LIN {X 0,Y 573.25,Z 579.072,A -85,B 0,C 180,E1 -2309.824,E2 -2309.824} C_VEL
LIN {X 0,Y 573.282,Z 579.069,A -85,B 0,C 180,E1 -2312.234,E2 -2312.234} C_VEL
LIN {X 0,Y 573.261,Z 579.079,A -85,B 0,C 180,E1 -2315.12,E2 -2315.12} C_VEL
LIN {X 0,Y 573.229,Z 579.076,A -85,B 0,C 180,E1 -2317.662,E2 -2317.662} C_VEL
LIN {X 0,Y 573.247,Z 579.073,A -85,B 0,C 180,E1 -2319.923,E2 -2319.923} C_VEL
LIN {X 0,Y 573.252,Z 579.08,A -85,B 0,C 180,E1 -2322.989,E2 -2322.989} C_VEL
LIN {X 0,Y 573.263,Z 579.072,A -85,B 0,C 180,E1 -2325.806,E2 -2325.806} C_VEL
LIN {X 0,Y 573.273,Z 579.072,A -85,B 0,C 180,E1 -2328.734,E2 -2328.734} C_VEL
LIN {X 0,Y 573.299,Z 579.072,A -85,B 0,C 180,E1 -2331.54,E2 -2331.54} C_VEL
LIN {X 0,Y 573.289,Z 579.067,A -85,B 0,C 180,E1 -2334.371,E2 -2334.371} C_VEL
LIN {X 0,Y 573.299,Z 579.069,A -85,B 0,C 180,E1 -2337.892,E2 -2337.892} C_VEL
LIN {X 0,Y 573.328,Z 579.063,A -85,B 0,C 180,E1 -2340.702,E2 -2340.702} C_VEL
LIN {X 0,Y 573.234,Z 579.085,A -85,B 0,C 180,E1 -2343.514,E2 -2343.514} C_VEL
LIN {X 0,Y 573.283,Z 579.078,A -85,B 0,C 180,E1 -2345.628,E2 -2345.628} C_VEL
LIN {X 0,Y 573.298,Z 579.066,A -85,B 0,C 180,E1 -2348.459,E2 -2348.459} C_VEL
LIN {X 0,Y 573.288,Z 579.072,A -85,B 0,C 180,E1 -2351.311,E2 -2351.311} C_VEL
LIN {X 0,Y 573.269,Z 579.07,A -85,B 0,C 180,E1 -2354.425,E2 -2354.425} C_VEL
LIN {X 0,Y 573.248,Z 579.073,A -85,B 0,C 180,E1 -2357.111,E2 -2357.111} C_VEL
LIN {X 0,Y 573.246,Z 579.079,A -85,B 0,C 180,E1 -2360.076,E2 -2360.076} C_VEL
LIN {X 0,Y 573.227,Z 579.078,A -85,B 0,C 180,E1 -2362.338,E2 -2362.338} C_VEL
LIN {X 0,Y 573.241,Z 579.076,A -85,B 0,C 180,E1 -2364.4,E2 -2364.4} C_VEL
LIN {X 0,Y 572.615,Z 579.154,A -85,B 0,C 180,E1 -2364.986,E2 -2364.986} C_VEL
LIN {X 0,Y 569.777,Z 579.515,A -85,B 0,C 180,E1 -2365.938,E2 -2365.938} C_VEL
LIN {X 0,Y 567.349,Z 579.813,A -85,B 0,C 180,E1 -2366.704,E2 -2366.704} C_VEL
LIN {X 0,Y 566.297,Z 579.94,A -85,B 0,C 180,E1 -2367.295,E2 -2367.295} C_VEL
LIN {X 0,Y 566.207,Z 579.951,A -85,B 0,C 180,E1 -2367.495,E2 -2367.495} C_VEL
LIN {X 0,Y 566.184,Z 579.954,A -85,B 0,C 180,E1 -2370.592,E2 -2370.592} C_VEL
LIN {X 0,Y 566.219,Z 579.948,A -85,B 0,C 180,E1 -2373.102,E2 -2373.102} C_VEL
LIN {X 0,Y 566.202,Z 579.954,A -85,B 0,C 180,E1 -2375.689,E2 -2375.689} C_VEL
LIN {X 0,Y 566.209,Z 579.953,A -85,B 0,C 180,E1 -2378.56,E2 -2378.56} C_VEL
LIN {X 0,Y 566.212,Z 579.949,A -85,B 0,C 180,E1 -2381.136,E2 -2381.136} C_VEL
LIN {X 0,Y 566.192,Z 579.958,A -85,B 0,C 180,E1 -2384.036,E2 -2384.036} C_VEL
LIN {X 0,Y 566.196,Z 579.951,A -85,B 0,C 180,E1 -2387.083,E2 -2387.083} C_VEL
LIN {X 0,Y 566.219,Z 579.95,A -85,B 0,C 180,E1 -2389.803,E2 -2389.803} C_VEL
LIN {X 0,Y 566.192,Z 579.958,A -85,B 0,C 180,E1 -2392.599,E2 -2392.599} C_VEL
LIN {X 0,Y 566.215,Z 579.949,A -85,B 0,C 180,E1 -2395.184,E2 -2395.184} C_VEL
LIN {X 0,Y 566.23,Z 579.947,A -85,B 0,C 180,E1 -2397.744,E2 -2397.744} C_VEL
LIN {X 0,Y 566.199,Z 579.957,A -85,B 0,C 180,E1 -2400.328,E2 -2400.328} C_VEL
LIN {X 0,Y 566.214,Z 579.958,A -85,B 0,C 180,E1 -2402.662,E2 -2402.662} C_VEL
LIN {X 0,Y 566.231,Z 579.95,A -85,B 0,C 180,E1 -2405.039,E2 -2405.039} C_VEL
LIN {X 0,Y 566.191,Z 579.954,A -85,B 0,C 180,E1 -2408.138,E2 -2408.138} C_VEL
LIN {X 0,Y 566.232,Z 579.955,A -85,B 0,C 180,E1 -2410.612,E2 -2410.612} C_VEL
LIN {X 0,Y 566.217,Z 579.95,A -85,B 0,C 180,E1 -2413.413,E2 -2413.413} C_VEL
LIN {X 0,Y 566.198,Z 579.954,A -85,B 0,C 180,E1 -2416.359,E2 -2416.359} C_VEL
LIN {X 0,Y 566.231,Z 579.953,A -85,B 0,C 180,E1 -2418.675,E2 -2418.675} C_VEL
LIN {X 0,Y 566.231,Z 579.949,A -85,B 0,C 180,E1 -2421.435,E2 -2421.435} C_VEL
LIN {X 0,Y 566.261,Z 579.944,A -85,B 0,C 180,E1 -2424.302,E2 -2424.302} C_VEL
LIN {X 0,Y 566.282,Z 579.94,A -85,B 0,C 180,E1 -2427.866,E2 -2427.866} C_VEL
LIN {X 0,Y 566.298,Z 579.942,A -85,B 0,C 180,E1 -2430.711,E2 -2430.711} C_VEL
LIN {X 0,Y 566.27,Z 579.947,A -85,B 0,C 180,E1 -2432.845,E2 -2432.845} C_VEL
LIN {X 0,Y 566.263,Z 579.945,A -85,B 0,C 180,E1 -2435.698,E2 -2435.698} C_VEL
LIN {X 0,Y 566.226,Z 579.948,A -85,B 0,C 180,E1 -2438.566,E2 -2438.566} C_VEL
LIN {X 0,Y 566.239,Z 579.953,A -85,B 0,C 180,E1 -2441.454,E2 -2441.454} C_VEL
LIN {X 0,Y 566.231,Z 579.947,A -85,B 0,C 180,E1 -2444.507,E2 -2444.507} C_VEL
LIN {X 0,Y 566.201,Z 579.96,A -85,B 0,C 180,E1 -2447.331,E2 -2447.331} C_VEL
LIN {X 0,Y 566.21,Z 579.95,A -85,B 0,C 180,E1 -2450.337,E2 -2450.337} C_VEL
LIN {X 0,Y 566.185,Z 579.962,A -85,B 0,C 180,E1 -2453.403,E2 -2453.403} C_VEL
LIN {X 0,Y 566.22,Z 579.958,A -85,B 0,C 180,E1 -2455.748,E2 -2455.748} C_VEL
LIN {X 0,Y 566.26,Z 580.088,A -85,B 0,C 180,E1 -2456.596,E2 -2456.596} C_VEL
LIN {X 0,Y 566.352,Z 587.078,A -85,B 0,C 180,E1 -2457.933,E2 -2457.933} C_VEL
LIN {X 0,Y 566.242,Z 601.154,A -85,B 0,C 180,E1 -2460.588,E2 -2460.588} C_VEL
LIN {X 0,Y 566.228,Z 603.568,A -85,B 0,C 180,E1 -2461.04,E2 -2461.04} C_VEL
LIN {X 0,Y 567.169,Z 609.752,A -85,B 0,C 180,E1 -2461.159,E2 -2461.159} C_VEL
LIN {X 0,Y 566.935,Z 710.865,A -85,B 0,C 180,E1 -2462.465,E2 -2462.465} C_VEL
LIN {X 0,Y 566.836,Z 724.501,A -85,B 0,C 180,E1 -2462.802,E2 -2462.802} C_VEL
LIN {X 0,Y 566.711,Z 737.49,A -85,B 0,C 180,E1 -2463.281,E2 -2463.281} C_VEL
LIN {X 0,Y 566.576,Z 749.083,A -85,B 0,C 180,E1 -2463.862,E2 -2463.862} C_VEL
LIN {X 0,Y 566.403,Z 760.435,A -85,B 0,C 180,E1 -2464.587,E2 -2464.587} C_VEL
LIN {X 0,Y 566.311,Z 770.741,A -85,B 0,C 180,E1 -2465.409,E2 -2465.409} C_VEL
LIN {X 0,Y 566.173,Z 780.385,A -85,B 0,C 180,E1 -2466.364,E2 -2466.364} C_VEL
LIN {X 0,Y 566.044,Z 789.413,A -85,B 0,C 180,E1 -2467.472,E2 -2467.472} C_VEL
LIN {X 0,Y 565.992,Z 796.322,A -85,B 0,C 180,E1 -2468.531,E2 -2468.531} C_VEL
LIN {X 0,Y 565.963,Z 802.163,A -85,B 0,C 180,E1 -2469.656,E2 -2469.656} C_VEL
LIN {X 0,Y 565.922,Z 806.612,A -85,B 0,C 180,E1 -2470.753,E2 -2470.753} C_VEL
LIN {X 0,Y 565.913,Z 810.603,A -85,B 0,C 180,E1 -2472.113,E2 -2472.113} C_VEL
LIN {X 0,Y 565.848,Z 812.476,A -85,B 0,C 180,E1 -2473.086,E2 -2473.086} C_VEL
LIN {X 0,Y 565.843,Z 813.61,A -85,B 0,C 180,E1 -2474.069,E2 -2474.069} C_VEL
LIN {X 0,Y 565.822,Z 813.999,A -85,B 0,C 180,E1 -2475.07,E2 -2475.07} C_VEL
LIN {X 0,Y 565.841,Z 813.567,A -85,B 0,C 180,E1 -2476.085,E2 -2476.085} C_VEL
LIN {X 0,Y 565.858,Z 812.295,A -85,B 0,C 180,E1 -2477.119,E2 -2477.119} C_VEL
LIN {X 0,Y 565.914,Z 810.124,A -85,B 0,C 180,E1 -2478.169,E2 -2478.169} C_VEL
LIN {X 0,Y 565.919,Z 806.927,A -85,B 0,C 180,E1 -2479.246,E2 -2479.246} C_VEL
LIN {X 0,Y 565.962,Z 802.575,A -85,B 0,C 180,E1 -2480.343,E2 -2480.343} C_VEL
LIN {X 0,Y 565.986,Z 796.831,A -85,B 0,C 180,E1 -2481.469,E2 -2481.469} C_VEL
LIN {X 0,Y 566.059,Z 789.431,A -85,B 0,C 180,E1 -2482.616,E2 -2482.616} C_VEL
LIN {X 0,Y 566.161,Z 781.206,A -85,B 0,C 180,E1 -2483.635,E2 -2483.635} C_VEL
LIN {X 0,Y 566.282,Z 772.717,A -85,B 0,C 180,E1 -2484.499,E2 -2484.499} C_VEL
LIN {X 0,Y 566.387,Z 763.144,A -85,B 0,C 180,E1 -2485.303,E2 -2485.303} C_VEL
LIN {X 0,Y 566.546,Z 751.86,A -85,B 0,C 180,E1 -2486.067,E2 -2486.067} C_VEL
LIN {X 0,Y 566.673,Z 739.534,A -85,B 0,C 180,E1 -2486.716,E2 -2486.716} C_VEL
LIN {X 0,Y 566.824,Z 727.276,A -85,B 0,C 180,E1 -2487.2,E2 -2487.2} C_VEL
LIN {X 0,Y 566.908,Z 714.232,A -85,B 0,C 180,E1 -2487.557,E2 -2487.557} C_VEL
LIN {X 0,Y 566.964,Z 698.519,A -85,B 0,C 180,E1 -2487.804,E2 -2487.804} C_VEL
LIN {X 0,Y 567.028,Z 608.635,A -85,B 0,C 180,E1 -2488.948,E2 -2488.948} C_VEL
LIN {X 0,Y 566.211,Z 603.648,A -85,B 0,C 180,E1 -2489.035,E2 -2489.035} C_VEL
LIN {X 0,Y 566.348,Z 589.127,A -85,B 0,C 180,E1 -2491.768,E2 -2491.768} C_VEL
LIN {X 0,Y 566.291,Z 580.244,A -85,B 0,C 180,E1 -2493.463,E2 -2493.463} C_VEL
LIN {X 0,Y 566.235,Z 579.952,A -85,B 0,C 180,E1 -2493.659,E2 -2493.659} C_VEL
LIN {X 0,Y 566.19,Z 579.955,A -85,B 0,C 180,E1 -2495.819,E2 -2495.819} C_VEL
LIN {X 0,Y 566.206,Z 579.956,A -85,B 0,C 180,E1 -2498.903,E2 -2498.903} C_VEL
LIN {X 0,Y 566.204,Z 579.953,A -85,B 0,C 180,E1 -2501.173,E2 -2501.173} C_VEL
LIN {X 0,Y 566.211,Z 579.95,A -85,B 0,C 180,E1 -2503.413,E2 -2503.413} C_VEL
LIN {X 0,Y 566.194,Z 579.957,A -85,B 0,C 180,E1 -2506.359,E2 -2506.359} C_VEL
LIN {X 0,Y 566.264,Z 579.953,A -85,B 0,C 180,E1 -2508.654,E2 -2508.654} C_VEL
LIN {X 0,Y 566.242,Z 579.947,A -85,B 0,C 180,E1 -2511.435,E2 -2511.435} C_VEL
LIN {X 0,Y 566.26,Z 579.946,A -85,B 0,C 180,E1 -2514.302,E2 -2514.302} C_VEL
LIN {X 0,Y 566.271,Z 579.942,A -85,B 0,C 180,E1 -2517.867,E2 -2517.867} C_VEL
LIN {X 0,Y 566.299,Z 579.946,A -85,B 0,C 180,E1 -2520.711,E2 -2520.711} C_VEL
LIN {X 0,Y 566.273,Z 579.951,A -85,B 0,C 180,E1 -2522.846,E2 -2522.846} C_VEL
LIN {X 0,Y 566.261,Z 579.944,A -85,B 0,C 180,E1 -2525.699,E2 -2525.699} C_VEL
LIN {X 0,Y 566.242,Z 579.949,A -85,B 0,C 180,E1 -2528.566,E2 -2528.566} C_VEL
LIN {X 0,Y 566.241,Z 579.949,A -85,B 0,C 180,E1 -2531.455,E2 -2531.455} C_VEL
LIN {X 0,Y 566.224,Z 579.95,A -85,B 0,C 180,E1 -2534.508,E2 -2534.508} C_VEL
LIN {X 0,Y 566.196,Z 579.958,A -85,B 0,C 180,E1 -2537.332,E2 -2537.332} C_VEL
LIN {X 0,Y 566.212,Z 579.949,A -85,B 0,C 180,E1 -2540.338,E2 -2540.338} C_VEL
LIN {X 0,Y 566.182,Z 579.959,A -85,B 0,C 180,E1 -2543.405,E2 -2543.405} C_VEL
LIN {X 0,Y 566.218,Z 579.95,A -85,B 0,C 180,E1 -2545.749,E2 -2545.749} C_VEL
LIN {X 0,Y 566.199,Z 579.95,A -85,B 0,C 180,E1 -2548.204,E2 -2548.204} C_VEL
LIN {X 0,Y 566.188,Z 579.953,A -85,B 0,C 180,E1 -2550.593,E2 -2550.593} C_VEL
LIN {X 0,Y 566.223,Z 579.953,A -85,B 0,C 180,E1 -2553.102,E2 -2553.102} C_VEL
LIN {X 0,Y 566.206,Z 579.954,A -85,B 0,C 180,E1 -2555.689,E2 -2555.689} C_VEL
LIN {X 0,Y 566.213,Z 579.949,A -85,B 0,C 180,E1 -2558.56,E2 -2558.56} C_VEL
LIN {X 0,Y 566.208,Z 579.955,A -85,B 0,C 180,E1 -2561.137,E2 -2561.137} C_VEL
LIN {X 0,Y 566.196,Z 579.953,A -85,B 0,C 180,E1 -2564.036,E2 -2564.036} C_VEL
LIN {X 0,Y 566.198,Z 579.955,A -85,B 0,C 180,E1 -2567.084,E2 -2567.084} C_VEL
LIN {X 0,Y 566.224,Z 579.954,A -85,B 0,C 180,E1 -2569.804,E2 -2569.804} C_VEL
LIN {X 0,Y 566.197,Z 579.951,A -85,B 0,C 180,E1 -2572.6,E2 -2572.6} C_VEL
LIN {X 0,Y 566.219,Z 579.952,A -85,B 0,C 180,E1 -2575.184,E2 -2575.184} C_VEL
LIN {X 0,Y 566.232,Z 579.956,A -85,B 0,C 180,E1 -2577.744,E2 -2577.744} C_VEL
LIN {X 0,Y 566.203,Z 579.953,A -85,B 0,C 180,E1 -2580.329,E2 -2580.329} C_VEL
LIN {X 0,Y 566.212,Z 579.951,A -85,B 0,C 180,E1 -2582.662,E2 -2582.662} C_VEL
LIN {X 0,Y 566.238,Z 579.95,A -85,B 0,C 180,E1 -2585.04,E2 -2585.04} C_VEL
LIN {X 0,Y 566.238,Z 579.992,A -85,B 0,C 180,E1 -2585.848,E2 -2585.848} C_VEL
LIN {X 0,Y 567.17,Z 585.129,A -85,B 0,C 180,E1 -2586.64,E2 -2586.64} C_VEL
LIN {X 0,Y 567.036,Z 601.083,A -85,B 0,C 180,E1 -2588.935,E2 -2588.935} C_VEL
LIN {X 0,Y 566.725,Z 622.357,A -85,B 0,C 180,E1 -2591.94,E2 -2591.94} C_VEL
LIN {X 0,Y 566.453,Z 642.3,A -85,B 0,C 180,E1 -2594.714,E2 -2594.714} C_VEL
LIN {X 0,Y 566.425,Z 651.524,A -85,B 0,C 180,E1 -2595.987,E2 -2595.987} C_VEL
LIN {X 0,Y 567.203,Z 658.268,A -85,B 0,C 180,E1 -2596.096,E2 -2596.096} C_VEL
LIN {X 0,Y 566.978,Z 759.962,A -85,B 0,C 180,E1 -2597.404,E2 -2597.404} C_VEL
LIN {X 0,Y 566.859,Z 772.467,A -85,B 0,C 180,E1 -2597.697,E2 -2597.697} C_VEL
LIN {X 0,Y 566.749,Z 785.381,A -85,B 0,C 180,E1 -2598.149,E2 -2598.149} C_VEL
LIN {X 0,Y 566.627,Z 797.158,A -85,B 0,C 180,E1 -2598.708,E2 -2598.708} C_VEL
LIN {X 0,Y 566.449,Z 809.206,A -85,B 0,C 180,E1 -2599.455,E2 -2599.455} C_VEL
LIN {X 0,Y 566.319,Z 819.603,A -85,B 0,C 180,E1 -2600.266,E2 -2600.266} C_VEL
LIN {X 0,Y 566.207,Z 828.115,A -85,B 0,C 180,E1 -2601.074,E2 -2601.074} C_VEL
LIN {X 0,Y 566.112,Z 835.962,A -85,B 0,C 180,E1 -2601.972,E2 -2601.972} C_VEL
LIN {X 0,Y 566.003,Z 843.622,A -85,B 0,C 180,E1 -2603.047,E2 -2603.047} C_VEL
LIN {X 0,Y 566.004,Z 850.681,A -85,B 0,C 180,E1 -2604.299,E2 -2604.299} C_VEL
LIN {X 0,Y 565.933,Z 855.372,A -85,B 0,C 180,E1 -2605.37,E2 -2605.37} C_VEL
LIN {X 0,Y 565.927,Z 858.957,A -85,B 0,C 180,E1 -2606.44,E2 -2606.44} C_VEL
LIN {X 0,Y 565.878,Z 860.808,A -85,B 0,C 180,E1 -2607.153,E2 -2607.153} C_VEL
LIN {X 0,Y 565.846,Z 863.186,A -85,B 0,C 180,E1 -2608.577,E2 -2608.577} C_VEL
LIN {X 0,Y 565.839,Z 864,A -85,B 0,C 180,E1 -2610,E2 -2610} C_VEL
LIN {X 0,Y 565.846,Z 863.186,A -85,B 0,C 180,E1 -2611.423,E2 -2611.423} C_VEL
LIN {X 0,Y 565.878,Z 860.81,A -85,B 0,C 180,E1 -2612.847,E2 -2612.847} C_VEL
LIN {X 0,Y 565.926,Z 857.896,A -85,B 0,C 180,E1 -2613.916,E2 -2613.916} C_VEL
LIN {X 0,Y 565.878,Z 853.95,A -85,B 0,C 180,E1 -2614.987,E2 -2614.987} C_VEL
LIN {X 0,Y 566.002,Z 848.867,A -85,B 0,C 180,E1 -2616.058,E2 -2616.058} C_VEL
LIN {X 0,Y 566.04,Z 842.47,A -85,B 0,C 180,E1 -2617.132,E2 -2617.132} C_VEL
LIN {X 0,Y 566.134,Z 834.48,A -85,B 0,C 180,E1 -2618.207,E2 -2618.207} C_VEL
LIN {X 0,Y 566.228,Z 826.338,A -85,B 0,C 180,E1 -2619.105,E2 -2619.105} C_VEL
LIN {X 0,Y 566.343,Z 816.404,A -85,B 0,C 180,E1 -2620.005,E2 -2620.005} C_VEL
LIN {X 0,Y 566.524,Z 805.293,A -85,B 0,C 180,E1 -2620.807,E2 -2620.807} C_VEL
LIN {X 0,Y 566.612,Z 794.183,A -85,B 0,C 180,E1 -2621.446,E2 -2621.446} C_VEL
LIN {X 0,Y 566.76,Z 781.992,A -85,B 0,C 180,E1 -2621.987,E2 -2621.987} C_VEL
LIN {X 0,Y 566.875,Z 769.189,A -85,B 0,C 180,E1 -2622.394,E2 -2622.394} C_VEL
LIN {X 0,Y 566.996,Z 755.622,A -85,B 0,C 180,E1 -2622.664,E2 -2622.664} C_VEL
LIN {X 0,Y 567.046,Z 655.806,A -85,B 0,C 180,E1 -2623.939,E2 -2623.939} C_VEL
LIN {X 0,Y 566.424,Z 651.441,A -85,B 0,C 180,E1 -2624.024,E2 -2624.024} C_VEL
LIN {X 0,Y 566.674,Z 627.675,A -85,B 0,C 180,E1 -2627.316,E2 -2627.316} C_VEL
LIN {X 0,Y 566.93,Z 607.733,A -85,B 0,C 180,E1 -2630.12,E2 -2630.12} C_VEL
LIN {X 0,Y 567.238,Z 587.788,A -85,B 0,C 180,E1 -2632.971,E2 -2632.971} C_VEL
LIN {X 0,Y 567.085,Z 584.236,A -85,B 0,C 180,E1 -2633.494,E2 -2633.494} C_VEL
LIN {X 0,Y 566.228,Z 579.955,A -85,B 0,C 180,E1 -2634.179,E2 -2634.179} C_VEL
LIN {X 0,Y 566.209,Z 579.956,A -85,B 0,C 180,E1 -2636.659,E2 -2636.659} C_VEL
LIN {X 0,Y 566.193,Z 579.954,A -85,B 0,C 180,E1 -2638.952,E2 -2638.952} C_VEL
LIN {X 0,Y 566.193,Z 579.952,A -85,B 0,C 180,E1 -2641.421,E2 -2641.421} C_VEL
LIN {X 0,Y 566.212,Z 579.952,A -85,B 0,C 180,E1 -2643.955,E2 -2643.955} C_VEL
LIN {X 0,Y 566.215,Z 579.958,A -85,B 0,C 180,E1 -2646.568,E2 -2646.568} C_VEL
LIN {X 0,Y 566.21,Z 579.949,A -85,B 0,C 180,E1 -2649.685,E2 -2649.685} C_VEL
LIN {X 0,Y 566.207,Z 579.952,A -85,B 0,C 180,E1 -2652.087,E2 -2652.087} C_VEL
LIN {X 0,Y 566.17,Z 579.958,A -85,B 0,C 180,E1 -2655.035,E2 -2655.035} C_VEL
LIN {X 0,Y 566.21,Z 579.949,A -85,B 0,C 180,E1 -2657.912,E2 -2657.912} C_VEL
LIN {X 0,Y 566.218,Z 579.959,A -85,B 0,C 180,E1 -2660.726,E2 -2660.726} C_VEL
LIN {X 0,Y 566.212,Z 579.949,A -85,B 0,C 180,E1 -2663.782,E2 -2663.782} C_VEL
LIN {X 0,Y 566.205,Z 579.951,A -85,B 0,C 180,E1 -2666.265,E2 -2666.265} C_VEL
LIN {X 0,Y 566.197,Z 579.961,A -85,B 0,C 180,E1 -2668.92,E2 -2668.92} C_VEL
LIN {X 0,Y 566.189,Z 579.96,A -85,B 0,C 180,E1 -2671.046,E2 -2671.046} C_VEL
LIN {X 0,Y 566.239,Z 579.948,A -85,B 0,C 180,E1 -2673.46,E2 -2673.46} C_VEL
LIN {X 0,Y 566.191,Z 579.952,A -85,B 0,C 180,E1 -2675.819,E2 -2675.819} C_VEL
LIN {X 0,Y 566.208,Z 579.957,A -85,B 0,C 180,E1 -2678.902,E2 -2678.902} C_VEL
LIN {X 0,Y 566.204,Z 579.96,A -85,B 0,C 180,E1 -2681.172,E2 -2681.172} C_VEL
LIN {X 0,Y 566.211,Z 579.955,A -85,B 0,C 180,E1 -2683.412,E2 -2683.412} C_VEL
LIN {X 0,Y 566.191,Z 579.952,A -85,B 0,C 180,E1 -2686.358,E2 -2686.358} C_VEL
LIN {X 0,Y 566.265,Z 579.944,A -85,B 0,C 180,E1 -2688.653,E2 -2688.653} C_VEL
LIN {X 0,Y 566.24,Z 579.953,A -85,B 0,C 180,E1 -2691.434,E2 -2691.434} C_VEL
LIN {X 0,Y 566.257,Z 579.943,A -85,B 0,C 180,E1 -2694.301,E2 -2694.301} C_VEL
LIN {X 0,Y 566.271,Z 579.945,A -85,B 0,C 180,E1 -2697.866,E2 -2697.866} C_VEL
LIN {X 0,Y 566.298,Z 579.939,A -85,B 0,C 180,E1 -2700.711,E2 -2700.711} C_VEL
LIN {X 0,Y 566.271,Z 579.943,A -85,B 0,C 180,E1 -2702.845,E2 -2702.845} C_VEL
LIN {X 0,Y 566.251,Z 579.952,A -85,B 0,C 180,E1 -2705.698,E2 -2705.698} C_VEL
LIN {X 0,Y 566.239,Z 579.945,A -85,B 0,C 180,E1 -2708.565,E2 -2708.565} C_VEL
LIN {X 0,Y 566.24,Z 579.952,A -85,B 0,C 180,E1 -2711.454,E2 -2711.454} C_VEL
LIN {X 0,Y 566.222,Z 579.948,A -85,B 0,C 180,E1 -2714.507,E2 -2714.507} C_VEL
LIN {X 0,Y 566.193,Z 579.955,A -85,B 0,C 180,E1 -2717.331,E2 -2717.331} C_VEL
LIN {X 0,Y 566.209,Z 579.952,A -85,B 0,C 180,E1 -2720.337,E2 -2720.337} C_VEL
LIN {X 0,Y 566.179,Z 579.956,A -85,B 0,C 180,E1 -2723.404,E2 -2723.404} C_VEL
LIN {X 0,Y 566.215,Z 579.956,A -85,B 0,C 180,E1 -2725.748,E2 -2725.748} C_VEL
LIN {X 0,Y 566.207,Z 579.951,A -85,B 0,C 180,E1 -2727.495,E2 -2727.495} C_VEL
LIN {X 0,Y 565.529,Z 580.042,A -85,B 0,C 180,E1 -2728.089,E2 -2728.089} C_VEL
LIN {X 0,Y 562.663,Z 580.397,A -85,B 0,C 180,E1 -2729.053,E2 -2729.053} C_VEL
LIN {X 0,Y 560.252,Z 580.699,A -85,B 0,C 180,E1 -2729.828,E2 -2729.828} C_VEL
LIN {X 0,Y 559.223,Z 580.823,A -85,B 0,C 180,E1 -2730.427,E2 -2730.427} C_VEL
LIN {X 0,Y 559.143,Z 580.831,A -85,B 0,C 180,E1 -2730.63,E2 -2730.63} C_VEL
LIN {X 0,Y 559.155,Z 580.831,A -85,B 0,C 180,E1 -2733.575,E2 -2733.575} C_VEL
LIN {X 0,Y 559.181,Z 580.829,A -85,B 0,C 180,E1 -2736.452,E2 -2736.452} C_VEL
LIN {X 0,Y 559.17,Z 580.826,A -85,B 0,C 180,E1 -2738.934,E2 -2738.934} C_VEL
LIN {X 0,Y 559.193,Z 580.826,A -85,B 0,C 180,E1 -2741.767,E2 -2741.767} C_VEL
LIN {X 0,Y 559.132,Z 580.834,A -85,B 0,C 180,E1 -2744.739,E2 -2744.739} C_VEL
LIN {X 0,Y 559.155,Z 580.828,A -85,B 0,C 180,E1 -2747.257,E2 -2747.257} C_VEL
LIN {X 0,Y 559.178,Z 580.832,A -85,B 0,C 180,E1 -2750.135,E2 -2750.135} C_VEL
LIN {X 0,Y 559.14,Z 580.833,A -85,B 0,C 180,E1 -2752.893,E2 -2752.893} C_VEL
LIN {X 0,Y 559.155,Z 580.828,A -85,B 0,C 180,E1 -2755.557,E2 -2755.557} C_VEL
LIN {X 0,Y 559.166,Z 580.831,A -85,B 0,C 180,E1 -2758.138,E2 -2758.138} C_VEL
LIN {X 0,Y 559.139,Z 580.839,A -85,B 0,C 180,E1 -2760.647,E2 -2760.647} C_VEL
LIN {X 0,Y 559.166,Z 580.828,A -85,B 0,C 180,E1 -2763.173,E2 -2763.173} C_VEL
LIN {X 0,Y 559.152,Z 580.828,A -85,B 0,C 180,E1 -2765.495,E2 -2765.495} C_VEL
LIN {X 0,Y 559.168,Z 580.836,A -85,B 0,C 180,E1 -2768.624,E2 -2768.624} C_VEL
LIN {X 0,Y 559.167,Z 580.834,A -85,B 0,C 180,E1 -2770.927,E2 -2770.927} C_VEL
LIN {X 0,Y 559.167,Z 580.827,A -85,B 0,C 180,E1 -2773.948,E2 -2773.948} C_VEL
LIN {X 0,Y 559.171,Z 580.827,A -85,B 0,C 180,E1 -2776.184,E2 -2776.184} C_VEL
LIN {X 0,Y 559.191,Z 580.83,A -85,B 0,C 180,E1 -2779.134,E2 -2779.134} C_VEL
LIN {X 0,Y 559.203,Z 580.822,A -85,B 0,C 180,E1 -2782.054,E2 -2782.054} C_VEL
LIN {X 0,Y 559.252,Z 580.826,A -85,B 0,C 180,E1 -2784.953,E2 -2784.953} C_VEL
LIN {X 0,Y 559.253,Z 580.816,A -85,B 0,C 180,E1 -2787.839,E2 -2787.839} C_VEL
LIN {X 0,Y 559.268,Z 580.818,A -85,B 0,C 180,E1 -2790.72,E2 -2790.72} C_VEL
LIN {X 0,Y 559.237,Z 580.824,A -85,B 0,C 180,E1 -2792.881,E2 -2792.881} C_VEL
LIN {X 0,Y 559.231,Z 580.82,A -85,B 0,C 180,E1 -2795.77,E2 -2795.77} C_VEL
LIN {X 0,Y 559.185,Z 580.826,A -85,B 0,C 180,E1 -2798.674,E2 -2798.674} C_VEL
LIN {X 0,Y 559.203,Z 580.827,A -85,B 0,C 180,E1 -2801.6,E2 -2801.6} C_VEL
LIN {X 0,Y 559.196,Z 580.823,A -85,B 0,C 180,E1 -2804.595,E2 -2804.595} C_VEL
LIN {X 0,Y 559.16,Z 580.835,A -85,B 0,C 180,E1 -2807.556,E2 -2807.556} C_VEL
LIN {X 0,Y 559.169,Z 580.831,A -85,B 0,C 180,E1 -2809.837,E2 -2809.837} C_VEL
LIN {X 0,Y 559.138,Z 580.832,A -85,B 0,C 180,E1 -2812.152,E2 -2812.152} C_VEL
LIN {X 0,Y 559.166,Z 580.833,A -85,B 0,C 180,E1 -2815.185,E2 -2815.185} C_VEL
LIN {X 0,Y 559.242,Z 580.929,A -85,B 0,C 180,E1 -2816.519,E2 -2816.519} C_VEL
LIN {X 0,Y 559.333,Z 588.875,A -85,B 0,C 180,E1 -2818.057,E2 -2818.057} C_VEL
LIN {X 0,Y 559.179,Z 603.564,A -85,B 0,C 180,E1 -2820.86,E2 -2820.86} C_VEL
LIN {X 0,Y 560.298,Z 611.174,A -85,B 0,C 180,E1 -2821.004,E2 -2821.004} C_VEL
LIN {X 0,Y 560.023,Z 710.413,A -85,B 0,C 180,E1 -2822.298,E2 -2822.298} C_VEL
LIN {X 0,Y 559.932,Z 723.682,A -85,B 0,C 180,E1 -2822.623,E2 -2822.623} C_VEL
LIN {X 0,Y 559.794,Z 736.752,A -85,B 0,C 180,E1 -2823.102,E2 -2823.102} C_VEL
LIN {X 0,Y 559.634,Z 747.407,A -85,B 0,C 180,E1 -2823.624,E2 -2823.624} C_VEL
LIN {X 0,Y 559.464,Z 758.28,A -85,B 0,C 180,E1 -2824.301,E2 -2824.301} C_VEL
LIN {X 0,Y 559.302,Z 769.442,A -85,B 0,C 180,E1 -2825.174,E2 -2825.174} C_VEL
LIN {X 0,Y 559.151,Z 778.983,A -85,B 0,C 180,E1 -2826.097,E2 -2826.097} C_VEL
LIN {X 0,Y 559.057,Z 787.471,A -85,B 0,C 180,E1 -2827.114,E2 -2827.114} C_VEL
LIN {X 0,Y 558.946,Z 794.928,A -85,B 0,C 180,E1 -2828.215,E2 -2828.215} C_VEL
LIN {X 0,Y 558.886,Z 801.419,A -85,B 0,C 180,E1 -2829.422,E2 -2829.422} C_VEL
LIN {X 0,Y 558.823,Z 805.408,A -85,B 0,C 180,E1 -2830.366,E2 -2830.366} C_VEL
LIN {X 0,Y 558.83,Z 808.779,A -85,B 0,C 180,E1 -2831.379,E2 -2831.379} C_VEL
LIN {X 0,Y 558.815,Z 810.654,A -85,B 0,C 180,E1 -2832.097,E2 -2832.097} C_VEL
LIN {X 0,Y 558.76,Z 812.619,A -85,B 0,C 180,E1 -2833.155,E2 -2833.155} C_VEL
LIN {X 0,Y 558.756,Z 813.703,A -85,B 0,C 180,E1 -2834.198,E2 -2834.198} C_VEL
LIN {X 0,Y 558.741,Z 813.968,A -85,B 0,C 180,E1 -2835.221,E2 -2835.221} C_VEL
LIN {X 0,Y 558.751,Z 813.464,A -85,B 0,C 180,E1 -2836.228,E2 -2836.228} C_VEL
LIN {X 0,Y 558.76,Z 812.18,A -85,B 0,C 180,E1 -2837.219,E2 -2837.219} C_VEL
LIN {X 0,Y 558.814,Z 810.148,A -85,B 0,C 180,E1 -2838.198,E2 -2838.198} C_VEL
LIN {X 0,Y 558.823,Z 807.407,A -85,B 0,C 180,E1 -2839.159,E2 -2839.159} C_VEL
LIN {X 0,Y 558.876,Z 802.873,A -85,B 0,C 180,E1 -2840.343,E2 -2840.343} C_VEL
LIN {X 0,Y 558.921,Z 796.567,A -85,B 0,C 180,E1 -2841.598,E2 -2841.598} C_VEL
LIN {X 0,Y 558.985,Z 789.999,A -85,B 0,C 180,E1 -2842.632,E2 -2842.632} C_VEL
LIN {X 0,Y 559.098,Z 781.814,A -85,B 0,C 180,E1 -2843.675,E2 -2843.675} C_VEL
LIN {X 0,Y 559.254,Z 772.012,A -85,B 0,C 180,E1 -2844.686,E2 -2844.686} C_VEL
LIN {X 0,Y 559.434,Z 761.253,A -85,B 0,C 180,E1 -2845.576,E2 -2845.576} C_VEL
LIN {X 0,Y 559.582,Z 750.402,A -85,B 0,C 180,E1 -2846.292,E2 -2846.292} C_VEL
LIN {X 0,Y 559.716,Z 737.959,A -85,B 0,C 180,E1 -2846.937,E2 -2846.937} C_VEL
LIN {X 0,Y 559.893,Z 724.987,A -85,B 0,C 180,E1 -2847.427,E2 -2847.427} C_VEL
LIN {X 0,Y 559.991,Z 711.747,A -85,B 0,C 180,E1 -2847.766,E2 -2847.766} C_VEL
LIN {X 0,Y 560.101,Z 683.414,A -85,B 0,C 180,E1 -2848.158,E2 -2848.158} C_VEL
LIN {X 0,Y 560.247,Z 610.136,A -85,B 0,C 180,E1 -2849.101,E2 -2849.101} C_VEL
LIN {X 0,Y 559.183,Z 603.625,A -85,B 0,C 180,E1 -2849.219,E2 -2849.219} C_VEL
LIN {X 0,Y 559.319,Z 589.349,A -85,B 0,C 180,E1 -2851.942,E2 -2851.942} C_VEL
LIN {X 0,Y 559.261,Z 581.26,A -85,B 0,C 180,E1 -2853.506,E2 -2853.506} C_VEL
LIN {X 0,Y 559.214,Z 580.827,A -85,B 0,C 180,E1 -2853.604,E2 -2853.604} C_VEL
LIN {X 0,Y 559.147,Z 580.84,A -85,B 0,C 180,E1 -2856.567,E2 -2856.567} C_VEL
LIN {X 0,Y 559.176,Z 580.827,A -85,B 0,C 180,E1 -2859.396,E2 -2859.396} C_VEL
LIN {X 0,Y 559.147,Z 580.83,A -85,B 0,C 180,E1 -2861.686,E2 -2861.686} C_VEL
LIN {X 0,Y 559.162,Z 580.829,A -85,B 0,C 180,E1 -2863.948,E2 -2863.948} C_VEL
LIN {X 0,Y 559.166,Z 580.83,A -85,B 0,C 180,E1 -2866.184,E2 -2866.184} C_VEL
LIN {X 0,Y 559.202,Z 580.827,A -85,B 0,C 180,E1 -2869.134,E2 -2869.134} C_VEL
LIN {X 0,Y 559.205,Z 580.824,A -85,B 0,C 180,E1 -2872.054,E2 -2872.054} C_VEL
LIN {X 0,Y 559.255,Z 580.824,A -85,B 0,C 180,E1 -2874.954,E2 -2874.954} C_VEL
LIN {X 0,Y 559.243,Z 580.818,A -85,B 0,C 180,E1 -2877.84,E2 -2877.84} C_VEL
LIN {X 0,Y 559.268,Z 580.822,A -85,B 0,C 180,E1 -2880.72,E2 -2880.72} C_VEL
LIN {X 0,Y 559.238,Z 580.828,A -85,B 0,C 180,E1 -2882.882,E2 -2882.882} C_VEL
LIN {X 0,Y 559.23,Z 580.819,A -85,B 0,C 180,E1 -2885.771,E2 -2885.771} C_VEL
LIN {X 0,Y 559.197,Z 580.828,A -85,B 0,C 180,E1 -2888.675,E2 -2888.675} C_VEL
LIN {X 0,Y 559.2,Z 580.825,A -85,B 0,C 180,E1 -2891.601,E2 -2891.601} C_VEL
LIN {X 0,Y 559.189,Z 580.827,A -85,B 0,C 180,E1 -2894.596,E2 -2894.596} C_VEL
LIN {X 0,Y 559.155,Z 580.832,A -85,B 0,C 180,E1 -2897.557,E2 -2897.557} C_VEL
LIN {X 0,Y 559.166,Z 580.828,A -85,B 0,C 180,E1 -2899.838,E2 -2899.838} C_VEL
LIN {X 0,Y 559.134,Z 580.83,A -85,B 0,C 180,E1 -2902.153,E2 -2902.153} C_VEL
LIN {X 0,Y 559.172,Z 580.835,A -85,B 0,C 180,E1 -2905.188,E2 -2905.188} C_VEL
LIN {X 0,Y 559.188,Z 580.826,A -85,B 0,C 180,E1 -2907.712,E2 -2907.712} C_VEL
LIN {X 0,Y 559.162,Z 580.827,A -85,B 0,C 180,E1 -2910.183,E2 -2910.183} C_VEL
LIN {X 0,Y 559.169,Z 580.827,A -85,B 0,C 180,E1 -2912.715,E2 -2912.715} C_VEL
LIN {X 0,Y 559.152,Z 580.837,A -85,B 0,C 180,E1 -2915.323,E2 -2915.323} C_VEL
LIN {X 0,Y 559.131,Z 580.832,A -85,B 0,C 180,E1 -2918.018,E2 -2918.018} C_VEL
LIN {X 0,Y 559.172,Z 580.828,A -85,B 0,C 180,E1 -2920.811,E2 -2920.811} C_VEL
LIN {X 0,Y 559.159,Z 580.834,A -85,B 0,C 180,E1 -2923.733,E2 -2923.733} C_VEL
LIN {X 0,Y 559.143,Z 580.831,A -85,B 0,C 180,E1 -2926.804,E2 -2926.804} C_VEL
LIN {X 0,Y 559.173,Z 580.831,A -85,B 0,C 180,E1 -2929.19,E2 -2929.19} C_VEL
LIN {X 0,Y 559.133,Z 580.835,A -85,B 0,C 180,E1 -2931.984,E2 -2931.984} C_VEL
LIN {X 0,Y 559.157,Z 580.829,A -85,B 0,C 180,E1 -2934.679,E2 -2934.679} C_VEL
LIN {X 0,Y 559.173,Z 580.833,A -85,B 0,C 180,E1 -2937.362,E2 -2937.362} C_VEL
LIN {X 0,Y 559.148,Z 580.833,A -85,B 0,C 180,E1 -2940.143,E2 -2940.143} C_VEL
LIN {X 0,Y 559.17,Z 580.83,A -85,B 0,C 180,E1 -2943.098,E2 -2943.098} C_VEL
LIN {X 0,Y 559.205,Z 580.989,A -85,B 0,C 180,E1 -2945.695,E2 -2945.695} C_VEL
LIN {X 0,Y 560.344,Z 587.788,A -85,B 0,C 180,E1 -2946.73,E2 -2946.73} C_VEL
LIN {X 0,Y 560.04,Z 606.402,A -85,B 0,C 180,E1 -2949.429,E2 -2949.429} C_VEL
LIN {X 0,Y 559.707,Z 626.345,A -85,B 0,C 180,E1 -2952.273,E2 -2952.273} C_VEL
LIN {X 0,Y 559.459,Z 646.292,A -85,B 0,C 180,E1 -2955.078,E2 -2955.078} C_VEL
LIN {X 0,Y 559.427,Z 651.524,A -85,B 0,C 180,E1 -2955.808,E2 -2955.808} C_VEL
LIN {X 0,Y 560.326,Z 658.268,A -85,B 0,C 180,E1 -2955.922,E2 -2955.922} C_VEL
LIN {X 0,Y 560.061,Z 759.962,A -85,B 0,C 180,E1 -2957.246,E2 -2957.246} C_VEL
LIN {X 0,Y 559.911,Z 772.467,A -85,B 0,C 180,E1 -2957.542,E2 -2957.542} C_VEL
LIN {X 0,Y 559.801,Z 785.383,A -85,B 0,C 180,E1 -2957.999,E2 -2957.999} C_VEL
LIN {X 0,Y 559.668,Z 796.815,A -85,B 0,C 180,E1 -2958.547,E2 -2958.547} C_VEL
LIN {X 0,Y 559.52,Z 807.913,A -85,B 0,C 180,E1 -2959.232,E2 -2959.232} C_VEL
LIN {X 0,Y 559.31,Z 818.543,A -85,B 0,C 180,E1 -2960.051,E2 -2960.051} C_VEL
LIN {X 0,Y 559.161,Z 828.115,A -85,B 0,C 180,E1 -2960.961,E2 -2960.961} C_VEL
LIN {X 0,Y 559.05,Z 835.962,A -85,B 0,C 180,E1 -2961.87,E2 -2961.87} C_VEL
LIN {X 0,Y 558.944,Z 843.623,A -85,B 0,C 180,E1 -2962.959,E2 -2962.959} C_VEL
LIN {X 0,Y 558.935,Z 850.681,A -85,B 0,C 180,E1 -2964.227,E2 -2964.227} C_VEL
LIN {X 0,Y 558.827,Z 855.373,A -85,B 0,C 180,E1 -2965.311,E2 -2965.311} C_VEL
LIN {X 0,Y 558.837,Z 858.958,A -85,B 0,C 180,E1 -2966.395,E2 -2966.395} C_VEL
LIN {X 0,Y 558.799,Z 860.808,A -85,B 0,C 180,E1 -2967.116,E2 -2967.116} C_VEL
LIN {X 0,Y 558.745,Z 863.185,A -85,B 0,C 180,E1 -2968.559,E2 -2968.559} C_VEL
LIN {X 0,Y 558.74,Z 864,A -85,B 0,C 180,E1 -2970,E2 -2970} C_VEL
LIN {X 0,Y 558.745,Z 863.186,A -85,B 0,C 180,E1 -2971.441,E2 -2971.441} C_VEL
LIN {X 0,Y 558.799,Z 860.81,A -85,B 0,C 180,E1 -2972.884,E2 -2972.884} C_VEL
LIN {X 0,Y 558.844,Z 857.896,A -85,B 0,C 180,E1 -2973.966,E2 -2973.966} C_VEL
LIN {X 0,Y 558.798,Z 853.949,A -85,B 0,C 180,E1 -2975.051,E2 -2975.051} C_VEL
LIN {X 0,Y 558.921,Z 848.868,A -85,B 0,C 180,E1 -2976.135,E2 -2976.135} C_VEL
LIN {X 0,Y 558.977,Z 842.469,A -85,B 0,C 180,E1 -2977.223,E2 -2977.223} C_VEL
LIN {X 0,Y 559.099,Z 834.48,A -85,B 0,C 180,E1 -2978.311,E2 -2978.311} C_VEL
LIN {X 0,Y 559.184,Z 826.338,A -85,B 0,C 180,E1 -2979.221,E2 -2979.221} C_VEL
LIN {X 0,Y 559.355,Z 816.404,A -85,B 0,C 180,E1 -2980.131,E2 -2980.131} C_VEL
LIN {X 0,Y 559.529,Z 805.401,A -85,B 0,C 180,E1 -2980.937,E2 -2980.937} C_VEL
LIN {X 0,Y 559.671,Z 793.468,A -85,B 0,C 180,E1 -2981.627,E2 -2981.627} C_VEL
LIN {X 0,Y 559.85,Z 780.776,A -85,B 0,C 180,E1 -2982.184,E2 -2982.184} C_VEL
LIN {X 0,Y 559.946,Z 767.36,A -85,B 0,C 180,E1 -2982.596,E2 -2982.596} C_VEL
LIN {X 0,Y 560.087,Z 754.107,A -85,B 0,C 180,E1 -2982.846,E2 -2982.846} C_VEL
LIN {X 0,Y 560.227,Z 657.211,A -85,B 0,C 180,E1 -2984.094,E2 -2984.094} C_VEL
LIN {X 0,Y 559.428,Z 651.441,A -85,B 0,C 180,E1 -2984.203,E2 -2984.203} C_VEL
LIN {X 0,Y 559.685,Z 628.794,A -85,B 0,C 180,E1 -2987.381,E2 -2987.381} C_VEL
LIN {X 0,Y 559.992,Z 609.061,A -85,B 0,C 180,E1 -2990.189,E2 -2990.189} C_VEL
LIN {X 0,Y 560.34,Z 589.117,A -85,B 0,C 180,E1 -2993.075,E2 -2993.075} C_VEL
LIN {X 0,Y 560.072,Z 585.113,A -85,B 0,C 180,E1 -2993.674,E2 -2993.674} C_VEL
LIN {X 0,Y 559.193,Z 580.832,A -85,B 0,C 180,E1 -2994.354,E2 -2994.354} C_VEL
LIN {X 0,Y 559.17,Z 580.83,A -85,B 0,C 180,E1 -2996.902,E2 -2996.902} C_VEL
LIN {X 0,Y 559.148,Z 580.833,A -85,B 0,C 180,E1 -2999.857,E2 -2999.857} C_VEL
LIN {X 0,Y 559.175,Z 580.831,A -85,B 0,C 180,E1 -3002.713,E2 -3002.713} C_VEL
LIN {X 0,Y 559.157,Z 580.828,A -85,B 0,C 180,E1 -3005.321,E2 -3005.321} C_VEL
LIN {X 0,Y 559.133,Z 580.833,A -85,B 0,C 180,E1 -3008.016,E2 -3008.016} C_VEL
LIN {X 0,Y 559.173,Z 580.832,A -85,B 0,C 180,E1 -3010.81,E2 -3010.81} C_VEL
LIN {X 0,Y 559.137,Z 580.83,A -85,B 0,C 180,E1 -3013.733,E2 -3013.733} C_VEL
LIN {X 0,Y 559.164,Z 580.835,A -85,B 0,C 180,E1 -3016.8,E2 -3016.8} C_VEL
LIN {X 0,Y 559.172,Z 580.829,A -85,B 0,C 180,E1 -3019.189,E2 -3019.189} C_VEL
LIN {X 0,Y 559.131,Z 580.831,A -85,B 0,C 180,E1 -3021.982,E2 -3021.982} C_VEL
LIN {X 0,Y 559.153,Z 580.838,A -85,B 0,C 180,E1 -3024.782,E2 -3024.782} C_VEL
LIN {X 0,Y 559.168,Z 580.829,A -85,B 0,C 180,E1 -3027.36,E2 -3027.36} C_VEL
LIN {X 0,Y 559.182,Z 580.825,A -85,B 0,C 180,E1 -3030.134,E2 -3030.134} C_VEL
LIN {X 0,Y 559.176,Z 580.832,A -85,B 0,C 180,E1 -3033.169,E2 -3033.169} C_VEL
LIN {X 0,Y 559.149,Z 580.832,A -85,B 0,C 180,E1 -3035.494,E2 -3035.494} C_VEL
LIN {X 0,Y 559.168,Z 580.83,A -85,B 0,C 180,E1 -3038.623,E2 -3038.623} C_VEL
LIN {X 0,Y 559.163,Z 580.834,A -85,B 0,C 180,E1 -3040.926,E2 -3040.926} C_VEL
LIN {X 0,Y 559.161,Z 580.828,A -85,B 0,C 180,E1 -3043.947,E2 -3043.947} C_VEL
LIN {X 0,Y 559.164,Z 580.827,A -85,B 0,C 180,E1 -3046.184,E2 -3046.184} C_VEL
LIN {X 0,Y 559.202,Z 580.83,A -85,B 0,C 180,E1 -3049.133,E2 -3049.133} C_VEL
LIN {X 0,Y 559.201,Z 580.823,A -85,B 0,C 180,E1 -3052.053,E2 -3052.053} C_VEL
LIN {X 0,Y 559.253,Z 580.819,A -85,B 0,C 180,E1 -3054.953,E2 -3054.953} C_VEL
LIN {X 0,Y 559.242,Z 580.821,A -85,B 0,C 180,E1 -3057.839,E2 -3057.839} C_VEL
LIN {X 0,Y 559.268,Z 580.815,A -85,B 0,C 180,E1 -3060.72,E2 -3060.72} C_VEL
LIN {X 0,Y 559.237,Z 580.819,A -85,B 0,C 180,E1 -3062.881,E2 -3062.881} C_VEL
LIN {X 0,Y 559.22,Z 580.827,A -85,B 0,C 180,E1 -3065.77,E2 -3065.77} C_VEL
LIN {X 0,Y 559.194,Z 580.823,A -85,B 0,C 180,E1 -3068.674,E2 -3068.674} C_VEL
LIN {X 0,Y 559.198,Z 580.832,A -85,B 0,C 180,E1 -3071.6,E2 -3071.6} C_VEL
LIN {X 0,Y 559.188,Z 580.824,A -85,B 0,C 180,E1 -3074.595,E2 -3074.595} C_VEL
LIN {X 0,Y 559.153,Z 580.835,A -85,B 0,C 180,E1 -3077.557,E2 -3077.557} C_VEL
LIN {X 0,Y 559.164,Z 580.837,A -85,B 0,C 180,E1 -3079.837,E2 -3079.837} C_VEL
LIN {X 0,Y 559.131,Z 580.836,A -85,B 0,C 180,E1 -3082.153,E2 -3082.153} C_VEL
LIN {X 0,Y 559.168,Z 580.827,A -85,B 0,C 180,E1 -3085.187,E2 -3085.187} C_VEL
LIN {X 0,Y 559.185,Z 580.83,A -85,B 0,C 180,E1 -3087.711,E2 -3087.711} C_VEL
LIN {X 0,Y 559.143,Z 580.831,A -85,B 0,C 180,E1 -3090.63,E2 -3090.63} C_VEL
LIN {X 0,Y 558.479,Z 580.913,A -85,B 0,C 180,E1 -3091.231,E2 -3091.231} C_VEL
LIN {X 0,Y 555.614,Z 581.276,A -85,B 0,C 180,E1 -3092.207,E2 -3092.207} C_VEL
LIN {X 0,Y 553.2,Z 581.573,A -85,B 0,C 180,E1 -3092.993,E2 -3092.993} C_VEL
LIN {X 0,Y 552.179,Z 581.7,A -85,B 0,C 180,E1 -3093.6,E2 -3093.6} C_VEL
LIN {X 0,Y 552.105,Z 581.712,A -85,B 0,C 180,E1 -3093.805,E2 -3093.805} C_VEL
LIN {X 0,Y 552.108,Z 581.707,A -85,B 0,C 180,E1 -3096.746,E2 -3096.746} C_VEL
LIN {X 0,Y 552.126,Z 581.705,A -85,B 0,C 180,E1 -3099.527,E2 -3099.527} C_VEL
LIN {X 0,Y 552.163,Z 581.699,A -85,B 0,C 180,E1 -3101.441,E2 -3101.441} C_VEL
LIN {X 0,Y 552.088,Z 581.714,A -85,B 0,C 180,E1 -3104.532,E2 -3104.532} C_VEL
LIN {X 0,Y 552.123,Z 581.705,A -85,B 0,C 180,E1 -3107.585,E2 -3107.585} C_VEL
LIN {X 0,Y 552.127,Z 581.712,A -85,B 0,C 180,E1 -3110.474,E2 -3110.474} C_VEL
LIN {X 0,Y 552.108,Z 581.706,A -85,B 0,C 180,E1 -3113.316,E2 -3113.316} C_VEL
LIN {X 0,Y 552.134,Z 581.705,A -85,B 0,C 180,E1 -3115.941,E2 -3115.941} C_VEL
LIN {X 0,Y 552.113,Z 581.715,A -85,B 0,C 180,E1 -3118.541,E2 -3118.541} C_VEL
LIN {X 0,Y 552.121,Z 581.704,A -85,B 0,C 180,E1 -3121.438,E2 -3121.438} C_VEL
LIN {X 0,Y 552.125,Z 581.709,A -85,B 0,C 180,E1 -3124.356,E2 -3124.356} C_VEL
LIN {X 0,Y 552.106,Z 581.715,A -85,B 0,C 180,E1 -3126.759,E2 -3126.759} C_VEL
LIN {X 0,Y 552.117,Z 581.708,A -85,B 0,C 180,E1 -3129.12,E2 -3129.12} C_VEL
LIN {X 0,Y 552.127,Z 581.704,A -85,B 0,C 180,E1 -3131.445,E2 -3131.445} C_VEL
LIN {X 0,Y 552.117,Z 581.705,A -85,B 0,C 180,E1 -3133.738,E2 -3133.738} C_VEL
LIN {X 0,Y 552.134,Z 581.703,A -85,B 0,C 180,E1 -3136.005,E2 -3136.005} C_VEL
LIN {X 0,Y 552.159,Z 581.708,A -85,B 0,C 180,E1 -3138.994,E2 -3138.994} C_VEL
LIN {X 0,Y 552.157,Z 581.7,A -85,B 0,C 180,E1 -3141.952,E2 -3141.952} C_VEL
LIN {X 0,Y 552.227,Z 581.7,A -85,B 0,C 180,E1 -3144.889,E2 -3144.889} C_VEL
LIN {X 0,Y 552.224,Z 581.692,A -85,B 0,C 180,E1 -3147.812,E2 -3147.812} C_VEL
LIN {X 0,Y 552.239,Z 581.694,A -85,B 0,C 180,E1 -3150.729,E2 -3150.729} C_VEL
LIN {X 0,Y 552.204,Z 581.701,A -85,B 0,C 180,E1 -3152.918,E2 -3152.918} C_VEL
LIN {X 0,Y 552.199,Z 581.696,A -85,B 0,C 180,E1 -3155.844,E2 -3155.844} C_VEL
LIN {X 0,Y 552.156,Z 581.703,A -85,B 0,C 180,E1 -3158.785,E2 -3158.785} C_VEL
LIN {X 0,Y 552.16,Z 581.702,A -85,B 0,C 180,E1 -3161.75,E2 -3161.75} C_VEL
LIN {X 0,Y 552.133,Z 581.704,A -85,B 0,C 180,E1 -3164.748,E2 -3164.748} C_VEL
LIN {X 0,Y 552.111,Z 581.709,A -85,B 0,C 180,E1 -3167.788,E2 -3167.788} C_VEL
LIN {X 0,Y 552.127,Z 581.706,A -85,B 0,C 180,E1 -3170.101,E2 -3170.101} C_VEL
LIN {X 0,Y 552.092,Z 581.709,A -85,B 0,C 180,E1 -3172.45,E2 -3172.45} C_VEL
LIN {X 0,Y 552.127,Z 581.713,A -85,B 0,C 180,E1 -3175.345,E2 -3175.345} C_VEL
LIN {X 0,Y 552.182,Z 581.839,A -85,B 0,C 180,E1 -3176.453,E2 -3176.453} C_VEL
LIN {X 0,Y 552.324,Z 586.993,A -85,B 0,C 180,E1 -3177.468,E2 -3177.468} C_VEL
LIN {X 0,Y 552.205,Z 600.401,A -85,B 0,C 180,E1 -3180.067,E2 -3180.067} C_VEL
LIN {X 0,Y 552.146,Z 603.617,A -85,B 0,C 180,E1 -3180.685,E2 -3180.685} C_VEL
LIN {X 0,Y 553.381,Z 610.877,A -85,B 0,C 180,E1 -3180.821,E2 -3180.821} C_VEL
LIN {X 0,Y 553.101,Z 709.968,A -85,B 0,C 180,E1 -3182.127,E2 -3182.127} C_VEL
LIN {X 0,Y 552.981,Z 723.201,A -85,B 0,C 180,E1 -3182.45,E2 -3182.45} C_VEL
LIN {X 0,Y 552.806,Z 735.388,A -85,B 0,C 180,E1 -3182.891,E2 -3182.891} C_VEL
LIN {X 0,Y 552.659,Z 747.349,A -85,B 0,C 180,E1 -3183.475,E2 -3183.475} C_VEL
LIN {X 0,Y 552.45,Z 759.057,A -85,B 0,C 180,E1 -3184.219,E2 -3184.219} C_VEL
LIN {X 0,Y 552.256,Z 770.32,A -85,B 0,C 180,E1 -3185.124,E2 -3185.124} C_VEL
LIN {X 0,Y 552.107,Z 779.728,A -85,B 0,C 180,E1 -3186.066,E2 -3186.066} C_VEL
LIN {X 0,Y 551.947,Z 788.959,A -85,B 0,C 180,E1 -3187.215,E2 -3187.215} C_VEL
LIN {X 0,Y 551.858,Z 796.565,A -85,B 0,C 180,E1 -3188.407,E2 -3188.407} C_VEL
LIN {X 0,Y 551.785,Z 802.335,A -85,B 0,C 180,E1 -3189.556,E2 -3189.556} C_VEL
LIN {X 0,Y 551.727,Z 807.461,A -85,B 0,C 180,E1 -3190.894,E2 -3190.894} C_VEL
LIN {X 0,Y 551.74,Z 810.316,A -85,B 0,C 180,E1 -3191.919,E2 -3191.919} C_VEL
LIN {X 0,Y 551.688,Z 811.495,A -85,B 0,C 180,E1 -3192.466,E2 -3192.466} C_VEL
LIN {X 0,Y 551.66,Z 813.056,A -85,B 0,C 180,E1 -3193.466,E2 -3193.466} C_VEL
LIN {X 0,Y 551.66,Z 813.883,A -85,B 0,C 180,E1 -3194.486,E2 -3194.486} C_VEL
LIN {X 0,Y 551.66,Z 813.904,A -85,B 0,C 180,E1 -3195.519,E2 -3195.519} C_VEL
LIN {X 0,Y 551.66,Z 813.12,A -85,B 0,C 180,E1 -3196.564,E2 -3196.564} C_VEL
LIN {X 0,Y 551.695,Z 811.476,A -85,B 0,C 180,E1 -3197.633,E2 -3197.633} C_VEL
LIN {X 0,Y 551.728,Z 808.878,A -85,B 0,C 180,E1 -3198.723,E2 -3198.723} C_VEL
LIN {X 0,Y 551.735,Z 805.19,A -85,B 0,C 180,E1 -3199.841,E2 -3199.841} C_VEL
LIN {X 0,Y 551.826,Z 799.244,A -85,B 0,C 180,E1 -3201.185,E2 -3201.185} C_VEL
LIN {X 0,Y 551.881,Z 792.737,A -85,B 0,C 180,E1 -3202.32,E2 -3202.32} C_VEL
LIN {X 0,Y 552.006,Z 785.561,A -85,B 0,C 180,E1 -3203.329,E2 -3203.329} C_VEL
LIN {X 0,Y 552.167,Z 776.373,A -85,B 0,C 180,E1 -3204.381,E2 -3204.381} C_VEL
LIN {X 0,Y 552.325,Z 766.921,A -85,B 0,C 180,E1 -3205.263,E2 -3205.263} C_VEL
LIN {X 0,Y 552.463,Z 756.154,A -85,B 0,C 180,E1 -3206.073,E2 -3206.073} C_VEL
LIN {X 0,Y 552.707,Z 743.874,A -85,B 0,C 180,E1 -3206.8,E2 -3206.8} C_VEL
LIN {X 0,Y 552.895,Z 731.52,A -85,B 0,C 180,E1 -3207.356,E2 -3207.356} C_VEL
LIN {X 0,Y 552.979,Z 718.07,A -85,B 0,C 180,E1 -3207.785,E2 -3207.785} C_VEL
LIN {X 0,Y 553.135,Z 706.033,A -85,B 0,C 180,E1 -3208.027,E2 -3208.027} C_VEL
LIN {X 0,Y 553.3,Z 610.239,A -85,B 0,C 180,E1 -3209.28,E2 -3209.28} C_VEL
LIN {X 0,Y 552.161,Z 603.569,A -85,B 0,C 180,E1 -3209.414,E2 -3209.414} C_VEL
LIN {X 0,Y 552.292,Z 589.578,A -85,B 0,C 180,E1 -3212.119,E2 -3212.119} C_VEL
LIN {X 0,Y 552.25,Z 582.268,A -85,B 0,C 180,E1 -3213.551,E2 -3213.551} C_VEL
LIN {X 0,Y 552.16,Z 581.706,A -85,B 0,C 180,E1 -3213.699,E2 -3213.699} C_VEL
LIN {X 0,Y 552.1,Z 581.716,A -85,B 0,C 180,E1 -3216.758,E2 -3216.758} C_VEL
LIN {X 0,Y 552.116,Z 581.708,A -85,B 0,C 180,E1 -3219.12,E2 -3219.12} C_VEL
LIN {X 0,Y 552.123,Z 581.706,A -85,B 0,C 180,E1 -3221.445,E2 -3221.445} C_VEL
LIN {X 0,Y 552.111,Z 581.706,A -85,B 0,C 180,E1 -3223.738,E2 -3223.738} C_VEL
LIN {X 0,Y 552.128,Z 581.705,A -85,B 0,C 180,E1 -3226.005,E2 -3226.005} C_VEL
LIN {X 0,Y 552.169,Z 581.705,A -85,B 0,C 180,E1 -3228.994,E2 -3228.994} C_VEL
LIN {X 0,Y 552.158,Z 581.701,A -85,B 0,C 180,E1 -3231.952,E2 -3231.952} C_VEL
LIN {X 0,Y 552.229,Z 581.701,A -85,B 0,C 180,E1 -3234.889,E2 -3234.889} C_VEL
LIN {X 0,Y 552.215,Z 581.693,A -85,B 0,C 180,E1 -3237.812,E2 -3237.812} C_VEL
LIN {X 0,Y 552.238,Z 581.698,A -85,B 0,C 180,E1 -3240.73,E2 -3240.73} C_VEL
LIN {X 0,Y 552.204,Z 581.704,A -85,B 0,C 180,E1 -3242.918,E2 -3242.918} C_VEL
LIN {X 0,Y 552.2,Z 581.695,A -85,B 0,C 180,E1 -3245.844,E2 -3245.844} C_VEL
LIN {X 0,Y 552.164,Z 581.706,A -85,B 0,C 180,E1 -3248.786,E2 -3248.786} C_VEL
LIN {X 0,Y 552.155,Z 581.701,A -85,B 0,C 180,E1 -3251.751,E2 -3251.751} C_VEL
LIN {X 0,Y 552.127,Z 581.709,A -85,B 0,C 180,E1 -3254.749,E2 -3254.749} C_VEL
LIN {X 0,Y 552.107,Z 581.708,A -85,B 0,C 180,E1 -3257.789,E2 -3257.789} C_VEL
LIN {X 0,Y 552.126,Z 581.704,A -85,B 0,C 180,E1 -3260.102,E2 -3260.102} C_VEL
LIN {X 0,Y 552.088,Z 581.709,A -85,B 0,C 180,E1 -3262.451,E2 -3262.451} C_VEL
LIN {X 0,Y 552.149,Z 581.708,A -85,B 0,C 180,E1 -3265.352,E2 -3265.352} C_VEL
LIN {X 0,Y 552.119,Z 581.704,A -85,B 0,C 180,E1 -3268.098,E2 -3268.098} C_VEL
LIN {X 0,Y 552.108,Z 581.707,A -85,B 0,C 180,E1 -3270.609,E2 -3270.609} C_VEL
LIN {X 0,Y 552.123,Z 581.711,A -85,B 0,C 180,E1 -3273.186,E2 -3273.186} C_VEL
LIN {X 0,Y 552.108,Z 581.709,A -85,B 0,C 180,E1 -3275.842,E2 -3275.842} C_VEL
LIN {X 0,Y 552.122,Z 581.709,A -85,B 0,C 180,E1 -3279.063,E2 -3279.063} C_VEL
LIN {X 0,Y 552.136,Z 581.712,A -85,B 0,C 180,E1 -3281.445,E2 -3281.445} C_VEL
LIN {X 0,Y 552.093,Z 581.709,A -85,B 0,C 180,E1 -3284.533,E2 -3284.533} C_VEL
LIN {X 0,Y 552.128,Z 581.713,A -85,B 0,C 180,E1 -3287.585,E2 -3287.585} C_VEL
LIN {X 0,Y 552.132,Z 581.704,A -85,B 0,C 180,E1 -3290.474,E2 -3290.474} C_VEL
LIN {X 0,Y 552.121,Z 581.711,A -85,B 0,C 180,E1 -3293.316,E2 -3293.316} C_VEL
LIN {X 0,Y 552.131,Z 581.71,A -85,B 0,C 180,E1 -3295.94,E2 -3295.94} C_VEL
LIN {X 0,Y 552.119,Z 581.705,A -85,B 0,C 180,E1 -3298.541,E2 -3298.541} C_VEL
LIN {X 0,Y 552.125,Z 581.712,A -85,B 0,C 180,E1 -3301.439,E2 -3301.439} C_VEL
LIN {X 0,Y 552.131,Z 581.709,A -85,B 0,C 180,E1 -3304.357,E2 -3304.357} C_VEL
LIN {X 0,Y 552.161,Z 581.862,A -85,B 0,C 180,E1 -3305.54,E2 -3305.54} C_VEL
LIN {X 0,Y 553.418,Z 589.157,A -85,B 0,C 180,E1 -3306.657,E2 -3306.657} C_VEL
LIN {X 0,Y 553.143,Z 606.402,A -85,B 0,C 180,E1 -3309.161,E2 -3309.161} C_VEL
LIN {X 0,Y 552.769,Z 626.345,A -85,B 0,C 180,E1 -3312.043,E2 -3312.043} C_VEL
LIN {X 0,Y 552.425,Z 647.753,A -85,B 0,C 180,E1 -3315.09,E2 -3315.09} C_VEL
LIN {X 0,Y 552.421,Z 651.535,A -85,B 0,C 180,E1 -3315.626,E2 -3315.626} C_VEL
LIN {X 0,Y 553.422,Z 659.753,A -85,B 0,C 180,E1 -3315.762,E2 -3315.762} C_VEL
LIN {X 0,Y 553.147,Z 759.962,A -85,B 0,C 180,E1 -3317.083,E2 -3317.083} C_VEL
LIN {X 0,Y 552.999,Z 772.466,A -85,B 0,C 180,E1 -3317.383,E2 -3317.383} C_VEL
LIN {X 0,Y 552.85,Z 785.376,A -85,B 0,C 180,E1 -3317.846,E2 -3317.846} C_VEL
LIN {X 0,Y 552.69,Z 797.669,A -85,B 0,C 180,E1 -3318.449,E2 -3318.449} C_VEL
LIN {X 0,Y 552.478,Z 809.202,A -85,B 0,C 180,E1 -3319.186,E2 -3319.186} C_VEL
LIN {X 0,Y 552.269,Z 819.605,A -85,B 0,C 180,E1 -3320.015,E2 -3320.015} C_VEL
LIN {X 0,Y 552.125,Z 828.115,A -85,B 0,C 180,E1 -3320.845,E2 -3320.845} C_VEL
LIN {X 0,Y 552.013,Z 835.962,A -85,B 0,C 180,E1 -3321.765,E2 -3321.765} C_VEL
LIN {X 0,Y 551.889,Z 843.622,A -85,B 0,C 180,E1 -3322.868,E2 -3322.868} C_VEL
LIN {X 0,Y 551.867,Z 850.68,A -85,B 0,C 180,E1 -3324.153,E2 -3324.153} C_VEL
LIN {X 0,Y 551.725,Z 855.373,A -85,B 0,C 180,E1 -3325.251,E2 -3325.251} C_VEL
LIN {X 0,Y 551.751,Z 858.958,A -85,B 0,C 180,E1 -3326.349,E2 -3326.349} C_VEL
LIN {X 0,Y 551.724,Z 860.808,A -85,B 0,C 180,E1 -3327.079,E2 -3327.079} C_VEL
LIN {X 0,Y 551.645,Z 863.185,A -85,B 0,C 180,E1 -3328.54,E2 -3328.54} C_VEL
LIN {X 0,Y 551.64,Z 864,A -85,B 0,C 180,E1 -3330,E2 -3330} C_VEL
LIN {X 0,Y 551.645,Z 863.186,A -85,B 0,C 180,E1 -3331.46,E2 -3331.46} C_VEL
LIN {X 0,Y 551.724,Z 860.81,A -85,B 0,C 180,E1 -3332.921,E2 -3332.921} C_VEL
LIN {X 0,Y 551.764,Z 857.896,A -85,B 0,C 180,E1 -3334.017,E2 -3334.017} C_VEL
LIN {X 0,Y 551.724,Z 853.949,A -85,B 0,C 180,E1 -3335.116,E2 -3335.116} C_VEL
LIN {X 0,Y 551.803,Z 848.192,A -85,B 0,C 180,E1 -3336.341,E2 -3336.341} C_VEL
LIN {X 0,Y 551.926,Z 841.238,A -85,B 0,C 180,E1 -3337.499,E2 -3337.499} C_VEL
LIN {X 0,Y 552.082,Z 832.993,A -85,B 0,C 180,E1 -3338.602,E2 -3338.602} C_VEL
LIN {X 0,Y 552.221,Z 824.541,A -85,B 0,C 180,E1 -3339.523,E2 -3339.523} C_VEL
LIN {X 0,Y 552.425,Z 814.099,A -85,B 0,C 180,E1 -3340.445,E2 -3340.445} C_VEL
LIN {X 0,Y 552.599,Z 803.294,A -85,B 0,C 180,E1 -3341.213,E2 -3341.213} C_VEL
LIN {X 0,Y 552.781,Z 792.414,A -85,B 0,C 180,E1 -3341.83,E2 -3341.83} C_VEL
LIN {X 0,Y 552.93,Z 780.772,A -85,B 0,C 180,E1 -3342.339,E2 -3342.339} C_VEL
LIN {X 0,Y 553.038,Z 767.359,A -85,B 0,C 180,E1 -3342.756,E2 -3342.756} C_VEL
LIN {X 0,Y 553.164,Z 754.107,A -85,B 0,C 180,E1 -3343.01,E2 -3343.01} C_VEL
LIN {X 0,Y 553.256,Z 657.182,A -85,B 0,C 180,E1 -3344.276,E2 -3344.276} C_VEL
LIN {X 0,Y 552.399,Z 651.451,A -85,B 0,C 180,E1 -3344.386,E2 -3344.386} C_VEL
LIN {X 0,Y 552.705,Z 629.488,A -85,B 0,C 180,E1 -3347.508,E2 -3347.508} C_VEL
LIN {X 0,Y 553.051,Z 610.391,A -85,B 0,C 180,E1 -3350.26,E2 -3350.26} C_VEL
LIN {X 0,Y 553.436,Z 590.28,A -85,B 0,C 180,E1 -3353.182,E2 -3353.182} C_VEL
LIN {X 0,Y 553.051,Z 586.155,A -85,B 0,C 180,E1 -3353.8,E2 -3353.8} C_VEL
LIN {X 0,Y 552.151,Z 581.71,A -85,B 0,C 180,E1 -3354.51,E2 -3354.51} C_VEL
LIN {X 0,Y 552.14,Z 581.704,A -85,B 0,C 180,E1 -3357.272,E2 -3357.272} C_VEL
LIN {X 0,Y 552.117,Z 581.711,A -85,B 0,C 180,E1 -3360.05,E2 -3360.05} C_VEL
LIN {X 0,Y 552.128,Z 581.707,A -85,B 0,C 180,E1 -3362.848,E2 -3362.848} C_VEL
LIN {X 0,Y 552.106,Z 581.706,A -85,B 0,C 180,E1 -3365.443,E2 -3365.443} C_VEL
LIN {X 0,Y 552.096,Z 581.709,A -85,B 0,C 180,E1 -3367.885,E2 -3367.885} C_VEL
LIN {X 0,Y 552.139,Z 581.711,A -85,B 0,C 180,E1 -3370.477,E2 -3370.477} C_VEL
LIN {X 0,Y 552.115,Z 581.705,A -85,B 0,C 180,E1 -3373.484,E2 -3373.484} C_VEL
LIN {X 0,Y 552.116,Z 581.714,A -85,B 0,C 180,E1 -3376.577,E2 -3376.577} C_VEL
LIN {X 0,Y 552.118,Z 581.705,A -85,B 0,C 180,E1 -3379.519,E2 -3379.519} C_VEL
LIN {X 0,Y 552.089,Z 581.711,A -85,B 0,C 180,E1 -3382.335,E2 -3382.335} C_VEL
LIN {X 0,Y 552.122,Z 581.71,A -85,B 0,C 180,E1 -3385.053,E2 -3385.053} C_VEL
LIN {X 0,Y 552.121,Z 581.704,A -85,B 0,C 180,E1 -3387.681,E2 -3387.681} C_VEL
LIN {X 0,Y 552.138,Z 581.703,A -85,B 0,C 180,E1 -3390.236,E2 -3390.236} C_VEL
LIN {X 0,Y 552.14,Z 581.712,A -85,B 0,C 180,E1 -3392.997,E2 -3392.997} C_VEL
LIN {X 0,Y 552.106,Z 581.714,A -85,B 0,C 180,E1 -3395.161,E2 -3395.161} C_VEL
LIN {X 0,Y 552.088,Z 581.711,A -85,B 0,C 180,E1 -3397.548,E2 -3397.548} C_VEL
LIN {X 0,Y 552.14,Z 581.703,A -85,B 0,C 180,E1 -3400.372,E2 -3400.372} C_VEL
LIN {X 0,Y 552.148,Z 581.708,A -85,B 0,C 180,E1 -3402.977,E2 -3402.977} C_VEL
LIN {X 0,Y 552.127,Z 581.704,A -85,B 0,C 180,E1 -3406.004,E2 -3406.004} C_VEL
LIN {X 0,Y 552.169,Z 581.704,A -85,B 0,C 180,E1 -3408.993,E2 -3408.993} C_VEL
LIN {X 0,Y 552.155,Z 581.701,A -85,B 0,C 180,E1 -3411.951,E2 -3411.951} C_VEL
LIN {X 0,Y 552.227,Z 581.694,A -85,B 0,C 180,E1 -3414.889,E2 -3414.889} C_VEL
LIN {X 0,Y 552.214,Z 581.696,A -85,B 0,C 180,E1 -3417.811,E2 -3417.811} C_VEL
LIN {X 0,Y 552.237,Z 581.69,A -85,B 0,C 180,E1 -3420.729,E2 -3420.729} C_VEL
LIN {X 0,Y 552.203,Z 581.696,A -85,B 0,C 180,E1 -3422.918,E2 -3422.918} C_VEL
LIN {X 0,Y 552.19,Z 581.701,A -85,B 0,C 180,E1 -3425.844,E2 -3425.844} C_VEL
LIN {X 0,Y 552.162,Z 581.699,A -85,B 0,C 180,E1 -3428.785,E2 -3428.785} C_VEL
LIN {X 0,Y 552.154,Z 581.709,A -85,B 0,C 180,E1 -3431.75,E2 -3431.75} C_VEL
LIN {X 0,Y 552.125,Z 581.704,A -85,B 0,C 180,E1 -3434.748,E2 -3434.748} C_VEL
LIN {X 0,Y 552.104,Z 581.717,A -85,B 0,C 180,E1 -3437.788,E2 -3437.788} C_VEL
LIN {X 0,Y 552.123,Z 581.709,A -85,B 0,C 180,E1 -3440.101,E2 -3440.101} C_VEL
LIN {X 0,Y 552.085,Z 581.71,A -85,B 0,C 180,E1 -3442.451,E2 -3442.451} C_VEL
LIN {X 0,Y 552.146,Z 581.703,A -85,B 0,C 180,E1 -3445.351,E2 -3445.351} C_VEL
LIN {X 0,Y 552.117,Z 581.713,A -85,B 0,C 180,E1 -3448.097,E2 -3448.097} C_VEL
LIN {X 0,Y 552.103,Z 581.708,A -85,B 0,C 180,E1 -3450.625,E2 -3450.625} C_VEL
LIN {X 0,Y 552.113,Z 581.705,A -85,B 0,C 180,E1 -3453.186,E2 -3453.186} C_VEL
LIN {X 0,Y 552.105,Z 581.712,A -85,B 0,C 180,E1 -3453.805,E2 -3453.805} C_VEL
LIN {X 0,Y 551.471,Z 581.797,A -85,B 0,C 180,E1 -3454.414,E2 -3454.414} C_VEL
LIN {X 0,Y 548.651,Z 582.147,A -85,B 0,C 180,E1 -3455.402,E2 -3455.402} C_VEL
LIN {X 0,Y 546.231,Z 582.447,A -85,B 0,C 180,E1 -3456.198,E2 -3456.198} C_VEL
LIN {X 0,Y 545.161,Z 582.573,A -85,B 0,C 180,E1 -3456.811,E2 -3456.811} C_VEL
LIN {X 0,Y 545.058,Z 582.584,A -85,B 0,C 180,E1 -3457.019,E2 -3457.019} C_VEL
LIN {X 0,Y 545.085,Z 582.59,A -85,B 0,C 180,E1 -3460.14,E2 -3460.14} C_VEL
LIN {X 0,Y 545.059,Z 582.587,A -85,B 0,C 180,E1 -3462.698,E2 -3462.698} C_VEL
LIN {X 0,Y 545.055,Z 582.585,A -85,B 0,C 180,E1 -3465.167,E2 -3465.167} C_VEL
LIN {X 0,Y 545.075,Z 582.585,A -85,B 0,C 180,E1 -3467.898,E2 -3467.898} C_VEL
LIN {X 0,Y 545.077,Z 582.585,A -85,B 0,C 180,E1 -3470.819,E2 -3470.819} C_VEL
LIN {X 0,Y 545.049,Z 582.586,A -85,B 0,C 180,E1 -3473.621,E2 -3473.621} C_VEL
LIN {X 0,Y 545.072,Z 582.59,A -85,B 0,C 180,E1 -3476.33,E2 -3476.33} C_VEL
LIN {X 0,Y 545.062,Z 582.587,A -85,B 0,C 180,E1 -3478.953,E2 -3478.953} C_VEL
LIN {X 0,Y 545.099,Z 582.579,A -85,B 0,C 180,E1 -3481.508,E2 -3481.508} C_VEL
LIN {X 0,Y 545.09,Z 582.588,A -85,B 0,C 180,E1 -3484.491,E2 -3484.491} C_VEL
LIN {X 0,Y 545.04,Z 582.588,A -85,B 0,C 180,E1 -3487.243,E2 -3487.243} C_VEL
LIN {X 0,Y 545.117,Z 582.582,A -85,B 0,C 180,E1 -3490.415,E2 -3490.415} C_VEL
LIN {X 0,Y 545.073,Z 582.583,A -85,B 0,C 180,E1 -3493.522,E2 -3493.522} C_VEL
LIN {X 0,Y 545.093,Z 582.58,A -85,B 0,C 180,E1 -3495.82,E2 -3495.82} C_VEL
LIN {X 0,Y 545.115,Z 582.587,A -85,B 0,C 180,E1 -3498.85,E2 -3498.85} C_VEL
LIN {X 0,Y 545.128,Z 582.575,A -85,B 0,C 180,E1 -3501.847,E2 -3501.847} C_VEL
LIN {X 0,Y 545.203,Z 582.573,A -85,B 0,C 180,E1 -3504.823,E2 -3504.823} C_VEL
LIN {X 0,Y 545.195,Z 582.568,A -85,B 0,C 180,E1 -3507.784,E2 -3507.784} C_VEL
LIN {X 0,Y 545.209,Z 582.57,A -85,B 0,C 180,E1 -3510.739,E2 -3510.739} C_VEL
LIN {X 0,Y 545.171,Z 582.577,A -85,B 0,C 180,E1 -3512.956,E2 -3512.956} C_VEL
LIN {X 0,Y 545.169,Z 582.571,A -85,B 0,C 180,E1 -3515.919,E2 -3515.919} C_VEL
LIN {X 0,Y 545.115,Z 582.581,A -85,B 0,C 180,E1 -3518.9,E2 -3518.9} C_VEL
LIN {X 0,Y 545.132,Z 582.576,A -85,B 0,C 180,E1 -3521.904,E2 -3521.904} C_VEL
LIN {X 0,Y 545.083,Z 582.585,A -85,B 0,C 180,E1 -3524.943,E2 -3524.943} C_VEL
LIN {X 0,Y 545.079,Z 582.583,A -85,B 0,C 180,E1 -3528.025,E2 -3528.025} C_VEL
LIN {X 0,Y 545.092,Z 582.581,A -85,B 0,C 180,E1 -3530.372,E2 -3530.372} C_VEL
LIN {X 0,Y 545.087,Z 582.591,A -85,B 0,C 180,E1 -3533.558,E2 -3533.558} C_VEL
LIN {X 0,Y 545.147,Z 582.639,A -85,B 0,C 180,E1 -3536.356,E2 -3536.356} C_VEL
LIN {X 0,Y 545.317,Z 587.808,A -85,B 0,C 180,E1 -3537.396,E2 -3537.396} C_VEL
LIN {X 0,Y 545.17,Z 602.002,A -85,B 0,C 180,E1 -3540.182,E2 -3540.182} C_VEL
LIN {X 0,Y 545.114,Z 603.639,A -85,B 0,C 180,E1 -3540.5,E2 -3540.5} C_VEL
LIN {X 0,Y 546.538,Z 613.023,A -85,B 0,C 180,E1 -3540.668,E2 -3540.668} C_VEL
LIN {X 0,Y 546.204,Z 710.282,A -85,B 0,C 180,E1 -3541.967,E2 -3541.967} C_VEL
LIN {X 0,Y 546.038,Z 723.551,A -85,B 0,C 180,E1 -3542.298,E2 -3542.298} C_VEL
LIN {X 0,Y 545.88,Z 735.341,A -85,B 0,C 180,E1 -3542.733,E2 -3542.733} C_VEL
LIN {X 0,Y 545.686,Z 747.561,A -85,B 0,C 180,E1 -3543.337,E2 -3543.337} C_VEL
LIN {X 0,Y 545.457,Z 759.18,A -85,B 0,C 180,E1 -3544.088,E2 -3544.088} C_VEL
LIN {X 0,Y 545.235,Z 770.385,A -85,B 0,C 180,E1 -3545.001,E2 -3545.001} C_VEL
LIN {X 0,Y 545.056,Z 780.192,A -85,B 0,C 180,E1 -3546.003,E2 -3546.003} C_VEL
LIN {X 0,Y 544.905,Z 788.728,A -85,B 0,C 180,E1 -3547.081,E2 -3547.081} C_VEL
LIN {X 0,Y 544.786,Z 796.226,A -85,B 0,C 180,E1 -3548.258,E2 -3548.258} C_VEL
LIN {X 0,Y 544.733,Z 801.427,A -85,B 0,C 180,E1 -3549.277,E2 -3549.277} C_VEL
LIN {X 0,Y 544.629,Z 806.055,A -85,B 0,C 180,E1 -3550.418,E2 -3550.418} C_VEL
LIN {X 0,Y 544.652,Z 809.521,A -85,B 0,C 180,E1 -3551.548,E2 -3551.548} C_VEL
LIN {X 0,Y 544.587,Z 811.903,A -85,B 0,C 180,E1 -3552.643,E2 -3552.643} C_VEL
LIN {X 0,Y 544.551,Z 813.705,A -85,B 0,C 180,E1 -3554.18,E2 -3554.18} C_VEL
LIN {X 0,Y 544.548,Z 813.969,A -85,B 0,C 180,E1 -3555.22,E2 -3555.22} C_VEL
LIN {X 0,Y 544.559,Z 813.444,A -85,B 0,C 180,E1 -3556.279,E2 -3556.279} C_VEL
LIN {X 0,Y 544.586,Z 812.057,A -85,B 0,C 180,E1 -3557.356,E2 -3557.356} C_VEL
LIN {X 0,Y 544.627,Z 808.67,A -85,B 0,C 180,E1 -3558.844,E2 -3558.844} C_VEL
LIN {X 0,Y 544.658,Z 805.501,A -85,B 0,C 180,E1 -3559.822,E2 -3559.822} C_VEL
LIN {X 0,Y 544.706,Z 800.41,A -85,B 0,C 180,E1 -3561.025,E2 -3561.025} C_VEL
LIN {X 0,Y 544.798,Z 793.519,A -85,B 0,C 180,E1 -3562.289,E2 -3562.289} C_VEL
LIN {X 0,Y 544.936,Z 786.205,A -85,B 0,C 180,E1 -3563.355,E2 -3563.355} C_VEL
LIN {X 0,Y 545.109,Z 777.576,A -85,B 0,C 180,E1 -3564.375,E2 -3564.375} C_VEL
LIN {X 0,Y 545.294,Z 767.544,A -85,B 0,C 180,E1 -3565.341,E2 -3565.341} C_VEL
LIN {X 0,Y 545.468,Z 757.36,A -85,B 0,C 180,E1 -3566.135,E2 -3566.135} C_VEL
LIN {X 0,Y 545.704,Z 746.053,A -85,B 0,C 180,E1 -3566.835,E2 -3566.835} C_VEL
LIN {X 0,Y 545.919,Z 733.537,A -85,B 0,C 180,E1 -3567.434,E2 -3567.434} C_VEL
LIN {X 0,Y 546.087,Z 720.5,A -85,B 0,C 180,E1 -3567.883,E2 -3567.883} C_VEL
LIN {X 0,Y 546.217,Z 707.989,A -85,B 0,C 180,E1 -3568.162,E2 -3568.162} C_VEL
LIN {X 0,Y 546.502,Z 611.755,A -85,B 0,C 180,E1 -3569.44,E2 -3569.44} C_VEL
LIN {X 0,Y 545.146,Z 603.573,A -85,B 0,C 180,E1 -3569.602,E2 -3569.602} C_VEL
LIN {X 0,Y 545.285,Z 589.525,A -85,B 0,C 180,E1 -3572.355,E2 -3572.355} C_VEL
LIN {X 0,Y 545.257,Z 583.312,A -85,B 0,C 180,E1 -3573.597,E2 -3573.597} C_VEL
LIN {X 0,Y 545.132,Z 582.582,A -85,B 0,C 180,E1 -3573.797,E2 -3573.797} C_VEL
LIN {X 0,Y 545.081,Z 582.591,A -85,B 0,C 180,E1 -3576.441,E2 -3576.441} C_VEL
LIN {X 0,Y 545.088,Z 582.582,A -85,B 0,C 180,E1 -3579.628,E2 -3579.628} C_VEL
LIN {X 0,Y 545.085,Z 582.59,A -85,B 0,C 180,E1 -3582.75,E2 -3582.75} C_VEL
LIN {X 0,Y 545.086,Z 582.582,A -85,B 0,C 180,E1 -3585.82,E2 -3585.82} C_VEL
LIN {X 0,Y 545.123,Z 582.586,A -85,B 0,C 180,E1 -3588.85,E2 -3588.85} C_VEL
LIN {X 0,Y 545.127,Z 582.577,A -85,B 0,C 180,E1 -3591.847,E2 -3591.847} C_VEL
LIN {X 0,Y 545.204,Z 582.576,A -85,B 0,C 180,E1 -3594.823,E2 -3594.823} C_VEL
LIN {X 0,Y 545.187,Z 582.569,A -85,B 0,C 180,E1 -3597.784,E2 -3597.784} C_VEL
LIN {X 0,Y 545.207,Z 582.574,A -85,B 0,C 180,E1 -3600.739,E2 -3600.739} C_VEL
LIN {X 0,Y 545.17,Z 582.579,A -85,B 0,C 180,E1 -3602.956,E2 -3602.956} C_VEL
LIN {X 0,Y 545.171,Z 582.57,A -85,B 0,C 180,E1 -3605.92,E2 -3605.92} C_VEL
LIN {X 0,Y 545.121,Z 582.586,A -85,B 0,C 180,E1 -3608.9,E2 -3608.9} C_VEL
LIN {X 0,Y 545.127,Z 582.576,A -85,B 0,C 180,E1 -3611.905,E2 -3611.905} C_VEL
LIN {X 0,Y 545.076,Z 582.59,A -85,B 0,C 180,E1 -3614.944,E2 -3614.944} C_VEL
LIN {X 0,Y 545.075,Z 582.583,A -85,B 0,C 180,E1 -3618.026,E2 -3618.026} C_VEL
LIN {X 0,Y 545.091,Z 582.581,A -85,B 0,C 180,E1 -3620.373,E2 -3620.373} C_VEL
LIN {X 0,Y 545.084,Z 582.585,A -85,B 0,C 180,E1 -3623.56,E2 -3623.56} C_VEL
LIN {X 0,Y 545.082,Z 582.581,A -85,B 0,C 180,E1 -3626.001,E2 -3626.001} C_VEL
LIN {X 0,Y 545.085,Z 582.583,A -85,B 0,C 180,E1 -3628.75,E2 -3628.75} C_VEL
LIN {X 0,Y 545.071,Z 582.585,A -85,B 0,C 180,E1 -3631.683,E2 -3631.683} C_VEL
LIN {X 0,Y 545.078,Z 582.582,A -85,B 0,C 180,E1 -3634.564,E2 -3634.564} C_VEL
LIN {X 0,Y 545.063,Z 582.593,A -85,B 0,C 180,E1 -3637.302,E2 -3637.302} C_VEL
LIN {X 0,Y 545.072,Z 582.583,A -85,B 0,C 180,E1 -3640.142,E2 -3640.142} C_VEL
LIN {X 0,Y 545.083,Z 582.586,A -85,B 0,C 180,E1 -3643.107,E2 -3643.107} C_VEL
LIN {X 0,Y 545.063,Z 582.585,A -85,B 0,C 180,E1 -3646.225,E2 -3646.225} C_VEL
LIN {X 0,Y 545.097,Z 582.582,A -85,B 0,C 180,E1 -3648.888,E2 -3648.888} C_VEL
LIN {X 0,Y 545.052,Z 582.593,A -85,B 0,C 180,E1 -3651.764,E2 -3651.764} C_VEL
LIN {X 0,Y 545.064,Z 582.585,A -85,B 0,C 180,E1 -3654.535,E2 -3654.535} C_VEL
LIN {X 0,Y 545.081,Z 582.587,A -85,B 0,C 180,E1 -3657.213,E2 -3657.213} C_VEL
LIN {X 0,Y 545.064,Z 582.592,A -85,B 0,C 180,E1 -3659.811,E2 -3659.811} C_VEL
LIN {X 0,Y 545.081,Z 582.585,A -85,B 0,C 180,E1 -3662.345,E2 -3662.345} C_VEL
LIN {X 0,Y 545.11,Z 582.701,A -85,B 0,C 180,E1 -3665.381,E2 -3665.381} C_VEL
LIN {X 0,Y 546.447,Z 589.941,A -85,B 0,C 180,E1 -3666.504,E2 -3666.504} C_VEL
LIN {X 0,Y 546.251,Z 604.89,A -85,B 0,C 180,E1 -3668.688,E2 -3668.688} C_VEL
LIN {X 0,Y 545.839,Z 626.345,A -85,B 0,C 180,E1 -3671.807,E2 -3671.807} C_VEL
LIN {X 0,Y 545.454,Z 647.619,A -85,B 0,C 180,E1 -3674.876,E2 -3674.876} C_VEL
LIN {X 0,Y 545.394,Z 651.526,A -85,B 0,C 180,E1 -3675.435,E2 -3675.435} C_VEL
LIN {X 0,Y 546.56,Z 660.608,A -85,B 0,C 180,E1 -3675.591,E2 -3675.591} C_VEL
LIN {X 0,Y 546.225,Z 759.962,A -85,B 0,C 180,E1 -3676.917,E2 -3676.917} C_VEL
LIN {X 0,Y 546.058,Z 773.228,A -85,B 0,C 180,E1 -3677.244,E2 -3677.244} C_VEL
LIN {X 0,Y 545.889,Z 786.495,A -85,B 0,C 180,E1 -3677.736,E2 -3677.736} C_VEL
LIN {X 0,Y 545.727,Z 798.372,A -85,B 0,C 180,E1 -3678.342,E2 -3678.342} C_VEL
LIN {X 0,Y 545.461,Z 810.489,A -85,B 0,C 180,E1 -3679.139,E2 -3679.139} C_VEL
LIN {X 0,Y 545.258,Z 820.649,A -85,B 0,C 180,E1 -3679.979,E2 -3679.979} C_VEL
LIN {X 0,Y 545.078,Z 829.788,A -85,B 0,C 180,E1 -3680.913,E2 -3680.913} C_VEL
LIN {X 0,Y 544.916,Z 838.69,A -85,B 0,C 180,E1 -3682.031,E2 -3682.031} C_VEL
LIN {X 0,Y 544.785,Z 845.85,A -85,B 0,C 180,E1 -3683.147,E2 -3683.147} C_VEL
LIN {X 0,Y 544.741,Z 852.367,A -85,B 0,C 180,E1 -3684.447,E2 -3684.447} C_VEL
LIN {X 0,Y 544.66,Z 856.677,A -85,B 0,C 180,E1 -3685.56,E2 -3685.56} C_VEL
LIN {X 0,Y 544.669,Z 858.958,A -85,B 0,C 180,E1 -3686.301,E2 -3686.301} C_VEL
LIN {X 0,Y 544.651,Z 860.808,A -85,B 0,C 180,E1 -3687.041,E2 -3687.041} C_VEL
LIN {X 0,Y 544.546,Z 863.184,A -85,B 0,C 180,E1 -3688.521,E2 -3688.521} C_VEL
LIN {X 0,Y 544.541,Z 864,A -85,B 0,C 180,E1 -3690,E2 -3690} C_VEL
LIN {X 0,Y 544.546,Z 863.185,A -85,B 0,C 180,E1 -3691.479,E2 -3691.479} C_VEL
LIN {X 0,Y 544.651,Z 860.81,A -85,B 0,C 180,E1 -3692.959,E2 -3692.959} C_VEL
LIN {X 0,Y 544.684,Z 857.896,A -85,B 0,C 180,E1 -3694.069,E2 -3694.069} C_VEL
LIN {X 0,Y 544.654,Z 853.949,A -85,B 0,C 180,E1 -3695.182,E2 -3695.182} C_VEL
LIN {X 0,Y 544.739,Z 848.706,A -85,B 0,C 180,E1 -3696.327,E2 -3696.327} C_VEL
LIN {X 0,Y 544.836,Z 842.469,A -85,B 0,C 180,E1 -3697.411,E2 -3697.411} C_VEL
LIN {X 0,Y 545.007,Z 834.479,A -85,B 0,C 180,E1 -3698.528,E2 -3698.528} C_VEL
LIN {X 0,Y 545.152,Z 826.336,A -85,B 0,C 180,E1 -3699.46,E2 -3699.46} C_VEL
LIN {X 0,Y 545.373,Z 816.402,A -85,B 0,C 180,E1 -3700.394,E2 -3700.394} C_VEL
LIN {X 0,Y 545.566,Z 805.598,A -85,B 0,C 180,E1 -3701.208,E2 -3701.208} C_VEL
LIN {X 0,Y 545.746,Z 794.179,A -85,B 0,C 180,E1 -3701.89,E2 -3701.89} C_VEL
LIN {X 0,Y 545.969,Z 781.983,A -85,B 0,C 180,E1 -3702.451,E2 -3702.451} C_VEL
LIN {X 0,Y 546.1,Z 769.187,A -85,B 0,C 180,E1 -3702.873,E2 -3702.873} C_VEL
LIN {X 0,Y 546.274,Z 755.622,A -85,B 0,C 180,E1 -3703.153,E2 -3703.153} C_VEL
LIN {X 0,Y 546.388,Z 657.797,A -85,B 0,C 180,E1 -3704.451,E2 -3704.451} C_VEL
LIN {X 0,Y 545.397,Z 651.491,A -85,B 0,C 180,E1 -3704.569,E2 -3704.569} C_VEL
LIN {X 0,Y 545.728,Z 630.184,A -85,B 0,C 180,E1 -3707.638,E2 -3707.638} C_VEL
LIN {X 0,Y 546.125,Z 610.321,A -85,B 0,C 180,E1 -3710.528,E2 -3710.528} C_VEL
LIN {X 0,Y 546.495,Z 591.363,A -85,B 0,C 180,E1 -3713.293,E2 -3713.293} C_VEL
LIN {X 0,Y 545.85,Z 586.199,A -85,B 0,C 180,E1 -3714.085,E2 -3714.085} C_VEL
LIN {X 0,Y 545.098,Z 582.588,A -85,B 0,C 180,E1 -3714.671,E2 -3714.671} C_VEL
LIN {X 0,Y 545.09,Z 582.584,A -85,B 0,C 180,E1 -3717.655,E2 -3717.655} C_VEL
LIN {X 0,Y 545.077,Z 582.591,A -85,B 0,C 180,E1 -3720.246,E2 -3720.246} C_VEL
LIN {X 0,Y 545.089,Z 582.582,A -85,B 0,C 180,E1 -3723.063,E2 -3723.063} C_VEL
LIN {X 0,Y 545.062,Z 582.584,A -85,B 0,C 180,E1 -3725.676,E2 -3725.676} C_VEL
LIN {X 0,Y 545.052,Z 582.59,A -85,B 0,C 180,E1 -3728.236,E2 -3728.236} C_VEL
LIN {X 0,Y 545.097,Z 582.581,A -85,B 0,C 180,E1 -3731.112,E2 -3731.112} C_VEL
LIN {X 0,Y 545.055,Z 582.587,A -85,B 0,C 180,E1 -3734.128,E2 -3734.128} C_VEL
LIN {X 0,Y 545.083,Z 582.588,A -85,B 0,C 180,E1 -3736.893,E2 -3736.893} C_VEL
LIN {X 0,Y 545.07,Z 582.583,A -85,B 0,C 180,E1 -3739.857,E2 -3739.857} C_VEL
LIN {X 0,Y 545.07,Z 582.588,A -85,B 0,C 180,E1 -3743.072,E2 -3743.072} C_VEL
LIN {X 0,Y 545.079,Z 582.582,A -85,B 0,C 180,E1 -3745.605,E2 -3745.605} C_VEL
LIN {X 0,Y 545.071,Z 582.584,A -85,B 0,C 180,E1 -3748.317,E2 -3748.317} C_VEL
LIN {X 0,Y 545.085,Z 582.586,A -85,B 0,C 180,E1 -3751.25,E2 -3751.25} C_VEL
LIN {X 0,Y 545.081,Z 582.581,A -85,B 0,C 180,E1 -3753.999,E2 -3753.999} C_VEL
LIN {X 0,Y 545.083,Z 582.583,A -85,B 0,C 180,E1 -3756.44,E2 -3756.44} C_VEL
LIN {X 0,Y 545.09,Z 582.582,A -85,B 0,C 180,E1 -3759.627,E2 -3759.627} C_VEL
LIN {X 0,Y 545.086,Z 582.584,A -85,B 0,C 180,E1 -3762.749,E2 -3762.749} C_VEL
LIN {X 0,Y 545.086,Z 582.582,A -85,B 0,C 180,E1 -3765.819,E2 -3765.819} C_VEL
LIN {X 0,Y 545.123,Z 582.58,A -85,B 0,C 180,E1 -3768.849,E2 -3768.849} C_VEL
LIN {X 0,Y 545.125,Z 582.578,A -85,B 0,C 180,E1 -3771.847,E2 -3771.847} C_VEL
LIN {X 0,Y 545.202,Z 582.568,A -85,B 0,C 180,E1 -3774.823,E2 -3774.823} C_VEL
LIN {X 0,Y 545.186,Z 582.572,A -85,B 0,C 180,E1 -3777.783,E2 -3777.783} C_VEL
LIN {X 0,Y 545.207,Z 582.566,A -85,B 0,C 180,E1 -3780.738,E2 -3780.738} C_VEL
LIN {X 0,Y 545.169,Z 582.572,A -85,B 0,C 180,E1 -3782.955,E2 -3782.955} C_VEL
LIN {X 0,Y 545.162,Z 582.576,A -85,B 0,C 180,E1 -3785.919,E2 -3785.919} C_VEL
LIN {X 0,Y 545.118,Z 582.577,A -85,B 0,C 180,E1 -3788.9,E2 -3788.9} C_VEL
LIN {X 0,Y 545.125,Z 582.582,A -85,B 0,C 180,E1 -3791.904,E2 -3791.904} C_VEL
LIN {X 0,Y 545.074,Z 582.582,A -85,B 0,C 180,E1 -3794.943,E2 -3794.943} C_VEL
LIN {X 0,Y 545.072,Z 582.588,A -85,B 0,C 180,E1 -3798.026,E2 -3798.026} C_VEL
LIN {X 0,Y 545.088,Z 582.582,A -85,B 0,C 180,E1 -3800.372,E2 -3800.372} C_VEL
LIN {X 0,Y 545.081,Z 582.586,A -85,B 0,C 180,E1 -3803.559,E2 -3803.559} C_VEL
LIN {X 0,Y 545.079,Z 582.591,A -85,B 0,C 180,E1 -3806,E2 -3806} C_VEL
LIN {X 0,Y 545.082,Z 582.582,A -85,B 0,C 180,E1 -3808.749,E2 -3808.749} C_VEL
LIN {X 0,Y 545.068,Z 582.587,A -85,B 0,C 180,E1 -3811.683,E2 -3811.683} C_VEL
LIN {X 0,Y 545.071,Z 582.585,A -85,B 0,C 180,E1 -3814.563,E2 -3814.563} C_VEL
LIN {X 0,Y 545.058,Z 582.584,A -85,B 0,C 180,E1 -3817.019,E2 -3817.019} C_VEL
LIN {X 0,Y 544.352,Z 582.676,A -85,B 0,C 180,E1 -3817.636,E2 -3817.636} C_VEL
LIN {X 0,Y 541.497,Z 583.03,A -85,B 0,C 180,E1 -3818.637,E2 -3818.637} C_VEL
LIN {X 0,Y 539.119,Z 583.326,A -85,B 0,C 180,E1 -3819.443,E2 -3819.443} C_VEL
LIN {X 0,Y 538.115,Z 583.457,A -85,B 0,C 180,E1 -3820.065,E2 -3820.065} C_VEL
LIN {X 0,Y 538.04,Z 583.459,A -85,B 0,C 180,E1 -3820.275,E2 -3820.275} C_VEL
LIN {X 0,Y 538.026,Z 583.461,A -85,B 0,C 180,E1 -3822.989,E2 -3822.989} C_VEL
LIN {X 0,Y 538.02,Z 583.465,A -85,B 0,C 180,E1 -3825.926,E2 -3825.926} C_VEL
LIN {X 0,Y 538.044,Z 583.458,A -85,B 0,C 180,E1 -3829.225,E2 -3829.225} C_VEL
LIN {X 0,Y 537.987,Z 583.47,A -85,B 0,C 180,E1 -3832.123,E2 -3832.123} C_VEL
LIN {X 0,Y 538.015,Z 583.464,A -85,B 0,C 180,E1 -3834.918,E2 -3834.918} C_VEL
LIN {X 0,Y 538.026,Z 583.46,A -85,B 0,C 180,E1 -3837.619,E2 -3837.619} C_VEL
LIN {X 0,Y 538.013,Z 583.467,A -85,B 0,C 180,E1 -3840.239,E2 -3840.239} C_VEL
LIN {X 0,Y 538.061,Z 583.462,A -85,B 0,C 180,E1 -3842.797,E2 -3842.797} C_VEL
LIN {X 0,Y 538.044,Z 583.459,A -85,B 0,C 180,E1 -3845.293,E2 -3845.293} C_VEL
LIN {X 0,Y 538.011,Z 583.463,A -85,B 0,C 180,E1 -3848.042,E2 -3848.042} C_VEL
LIN {X 0,Y 538.037,Z 583.465,A -85,B 0,C 180,E1 -3850.941,E2 -3850.941} C_VEL
LIN {X 0,Y 538.023,Z 583.463,A -85,B 0,C 180,E1 -3853.299,E2 -3853.299} C_VEL
LIN {X 0,Y 538.061,Z 583.456,A -85,B 0,C 180,E1 -3855.631,E2 -3855.631} C_VEL
LIN {X 0,Y 538.074,Z 583.461,A -85,B 0,C 180,E1 -3858.702,E2 -3858.702} C_VEL
LIN {X 0,Y 538.085,Z 583.453,A -85,B 0,C 180,E1 -3861.74,E2 -3861.74} C_VEL
LIN {X 0,Y 538.16,Z 583.45,A -85,B 0,C 180,E1 -3864.755,E2 -3864.755} C_VEL
LIN {X 0,Y 538.167,Z 583.443,A -85,B 0,C 180,E1 -3867.755,E2 -3867.755} C_VEL
LIN {X 0,Y 538.179,Z 583.445,A -85,B 0,C 180,E1 -3870.748,E2 -3870.748} C_VEL
LIN {X 0,Y 538.138,Z 583.454,A -85,B 0,C 180,E1 -3872.994,E2 -3872.994} C_VEL
LIN {X 0,Y 538.119,Z 583.449,A -85,B 0,C 180,E1 -3875.997,E2 -3875.997} C_VEL
LIN {X 0,Y 538.066,Z 583.461,A -85,B 0,C 180,E1 -3879.017,E2 -3879.017} C_VEL
LIN {X 0,Y 538.081,Z 583.454,A -85,B 0,C 180,E1 -3882.062,E2 -3882.062} C_VEL
LIN {X 0,Y 538.042,Z 583.465,A -85,B 0,C 180,E1 -3885.143,E2 -3885.143} C_VEL
LIN {X 0,Y 538.031,Z 583.46,A -85,B 0,C 180,E1 -3888.27,E2 -3888.27} C_VEL
LIN {X 0,Y 538.036,Z 583.461,A -85,B 0,C 180,E1 -3890.651,E2 -3890.651} C_VEL
LIN {X 0,Y 538.02,Z 583.468,A -85,B 0,C 180,E1 -3893.887,E2 -3893.887} C_VEL
LIN {X 0,Y 538.099,Z 583.61,A -85,B 0,C 180,E1 -3896.258,E2 -3896.258} C_VEL
LIN {X 0,Y 538.353,Z 588.087,A -85,B 0,C 180,E1 -3897.187,E2 -3897.187} C_VEL
LIN {X 0,Y 538.136,Z 602.425,A -85,B 0,C 180,E1 -3900.067,E2 -3900.067} C_VEL
LIN {X 0,Y 538.089,Z 603.64,A -85,B 0,C 180,E1 -3900.306,E2 -3900.306} C_VEL
LIN {X 0,Y 539.651,Z 614.067,A -85,B 0,C 180,E1 -3900.494,E2 -3900.494} C_VEL
LIN {X 0,Y 539.296,Z 710.714,A -85,B 0,C 180,E1 -3901.805,E2 -3901.805} C_VEL
LIN {X 0,Y 539.112,Z 724.375,A -85,B 0,C 180,E1 -3902.158,E2 -3902.158} C_VEL
LIN {X 0,Y 538.939,Z 737.189,A -85,B 0,C 180,E1 -3902.652,E2 -3902.652} C_VEL
LIN {X 0,Y 538.704,Z 748.263,A -85,B 0,C 180,E1 -3903.225,E2 -3903.225} C_VEL
LIN {X 0,Y 538.48,Z 759.048,A -85,B 0,C 180,E1 -3903.934,E2 -3903.934} C_VEL
LIN {X 0,Y 538.246,Z 769.955,A -85,B 0,C 180,E1 -3904.83,E2 -3904.83} C_VEL
LIN {X 0,Y 538.067,Z 778.798,A -85,B 0,C 180,E1 -3905.723,E2 -3905.723} C_VEL
LIN {X 0,Y 537.878,Z 786.83,A -85,B 0,C 180,E1 -3906.71,E2 -3906.71} C_VEL
LIN {X 0,Y 537.731,Z 794.654,A -85,B 0,C 180,E1 -3907.898,E2 -3907.898} C_VEL
LIN {X 0,Y 537.651,Z 801.402,A -85,B 0,C 180,E1 -3909.195,E2 -3909.195} C_VEL
LIN {X 0,Y 537.567,Z 805.7,A -85,B 0,C 180,E1 -3910.258,E2 -3910.258} C_VEL
LIN {X 0,Y 537.553,Z 809.014,A -85,B 0,C 180,E1 -3911.317,E2 -3911.317} C_VEL
LIN {X 0,Y 537.496,Z 812.257,A -85,B 0,C 180,E1 -3912.836,E2 -3912.836} C_VEL
LIN {X 0,Y 537.475,Z 813.607,A -85,B 0,C 180,E1 -3914.014,E2 -3914.014} C_VEL
LIN {X 0,Y 537.469,Z 813.998,A -85,B 0,C 180,E1 -3915.081,E2 -3915.081} C_VEL
LIN {X 0,Y 537.457,Z 813.573,A -85,B 0,C 180,E1 -3916.129,E2 -3916.129} C_VEL
LIN {X 0,Y 537.495,Z 812.39,A -85,B 0,C 180,E1 -3917.163,E2 -3917.163} C_VEL
LIN {X 0,Y 537.55,Z 809.268,A -85,B 0,C 180,E1 -3918.682,E2 -3918.682} C_VEL
LIN {X 0,Y 537.566,Z 806.029,A -85,B 0,C 180,E1 -3919.741,E2 -3919.741} C_VEL
LIN {X 0,Y 537.649,Z 801.803,A -85,B 0,C 180,E1 -3920.804,E2 -3920.804} C_VEL
LIN {X 0,Y 537.719,Z 796.479,A -85,B 0,C 180,E1 -3921.874,E2 -3921.874} C_VEL
LIN {X 0,Y 537.857,Z 789.15,A -85,B 0,C 180,E1 -3923.054,E2 -3923.054} C_VEL
LIN {X 0,Y 538,Z 781.22,A -85,B 0,C 180,E1 -3924.086,E2 -3924.086} C_VEL
LIN {X 0,Y 538.169,Z 772.218,A -85,B 0,C 180,E1 -3925.047,E2 -3925.047} C_VEL
LIN {X 0,Y 538.417,Z 761.694,A -85,B 0,C 180,E1 -3925.959,E2 -3925.959} C_VEL
LIN {X 0,Y 538.663,Z 751.109,A -85,B 0,C 180,E1 -3926.692,E2 -3926.692} C_VEL
LIN {X 0,Y 538.832,Z 739.279,A -85,B 0,C 180,E1 -3927.34,E2 -3927.34} C_VEL
LIN {X 0,Y 539.077,Z 726.482,A -85,B 0,C 180,E1 -3927.864,E2 -3927.864} C_VEL
LIN {X 0,Y 539.259,Z 713.73,A -85,B 0,C 180,E1 -3928.22,E2 -3928.22} C_VEL
LIN {X 0,Y 539.347,Z 697.441,A -85,B 0,C 180,E1 -3928.483,E2 -3928.483} C_VEL
LIN {X 0,Y 539.614,Z 612.35,A -85,B 0,C 180,E1 -3929.62,E2 -3929.62} C_VEL
LIN {X 0,Y 538.119,Z 603.592,A -85,B 0,C 180,E1 -3929.792,E2 -3929.792} C_VEL
LIN {X 0,Y 538.307,Z 591.037,A -85,B 0,C 180,E1 -3932.321,E2 -3932.321} C_VEL
LIN {X 0,Y 538.282,Z 584.623,A -85,B 0,C 180,E1 -3933.646,E2 -3933.646} C_VEL
LIN {X 0,Y 538.096,Z 583.459,A -85,B 0,C 180,E1 -3933.923,E2 -3933.923} C_VEL
LIN {X 0,Y 538.013,Z 583.468,A -85,B 0,C 180,E1 -3936.929,E2 -3936.929} C_VEL
LIN {X 0,Y 538.068,Z 583.459,A -85,B 0,C 180,E1 -3940.148,E2 -3940.148} C_VEL
LIN {X 0,Y 538.017,Z 583.464,A -85,B 0,C 180,E1 -3943.299,E2 -3943.299} C_VEL
LIN {X 0,Y 538.054,Z 583.458,A -85,B 0,C 180,E1 -3945.631,E2 -3945.631} C_VEL
LIN {X 0,Y 538.08,Z 583.464,A -85,B 0,C 180,E1 -3948.702,E2 -3948.702} C_VEL
LIN {X 0,Y 538.083,Z 583.454,A -85,B 0,C 180,E1 -3951.74,E2 -3951.74} C_VEL
LIN {X 0,Y 538.18,Z 583.45,A -85,B 0,C 180,E1 -3954.756,E2 -3954.756} C_VEL
LIN {X 0,Y 538.159,Z 583.445,A -85,B 0,C 180,E1 -3957.755,E2 -3957.755} C_VEL
LIN {X 0,Y 538.177,Z 583.45,A -85,B 0,C 180,E1 -3960.749,E2 -3960.749} C_VEL
LIN {X 0,Y 538.136,Z 583.455,A -85,B 0,C 180,E1 -3962.995,E2 -3962.995} C_VEL
LIN {X 0,Y 538.124,Z 583.448,A -85,B 0,C 180,E1 -3965.998,E2 -3965.998} C_VEL
LIN {X 0,Y 538.07,Z 583.463,A -85,B 0,C 180,E1 -3969.018,E2 -3969.018} C_VEL
LIN {X 0,Y 538.075,Z 583.454,A -85,B 0,C 180,E1 -3972.063,E2 -3972.063} C_VEL
LIN {X 0,Y 538.036,Z 583.467,A -85,B 0,C 180,E1 -3975.144,E2 -3975.144} C_VEL
LIN {X 0,Y 538.027,Z 583.461,A -85,B 0,C 180,E1 -3978.271,E2 -3978.271} C_VEL
LIN {X 0,Y 538.034,Z 583.462,A -85,B 0,C 180,E1 -3980.652,E2 -3980.652} C_VEL
LIN {X 0,Y 538.016,Z 583.463,A -85,B 0,C 180,E1 -3983.888,E2 -3983.888} C_VEL
LIN {X 0,Y 538.043,Z 583.457,A -85,B 0,C 180,E1 -3986.367,E2 -3986.367} C_VEL
LIN {X 0,Y 538.049,Z 583.462,A -85,B 0,C 180,E1 -3988.939,E2 -3988.939} C_VEL
LIN {X 0,Y 538.021,Z 583.461,A -85,B 0,C 180,E1 -3991.891,E2 -3991.891} C_VEL
LIN {X 0,Y 538.028,Z 583.46,A -85,B 0,C 180,E1 -3994.622,E2 -3994.622} C_VEL
LIN {X 0,Y 538.018,Z 583.468,A -85,B 0,C 180,E1 -3997.174,E2 -3997.174} C_VEL
LIN {X 0,Y 538.029,Z 583.464,A -85,B 0,C 180,E1 -3999.797,E2 -3999.797} C_VEL
LIN {X 0,Y 538.02,Z 583.463,A -85,B 0,C 180,E1 -4002.786,E2 -4002.786} C_VEL
LIN {X 0,Y 538.026,Z 583.464,A -85,B 0,C 180,E1 -4005.926,E2 -4005.926} C_VEL
LIN {X 0,Y 538.076,Z 583.46,A -85,B 0,C 180,E1 -4009.25,E2 -4009.25} C_VEL
LIN {X 0,Y 537.993,Z 583.468,A -85,B 0,C 180,E1 -4012.123,E2 -4012.123} C_VEL
LIN {X 0,Y 538.019,Z 583.463,A -85,B 0,C 180,E1 -4014.918,E2 -4014.918} C_VEL
LIN {X 0,Y 538.026,Z 583.471,A -85,B 0,C 180,E1 -4017.619,E2 -4017.619} C_VEL
LIN {X 0,Y 538.017,Z 583.465,A -85,B 0,C 180,E1 -4020.24,E2 -4020.24} C_VEL
LIN {X 0,Y 538.058,Z 583.459,A -85,B 0,C 180,E1 -4022.797,E2 -4022.797} C_VEL
LIN {X 0,Y 538.087,Z 583.567,A -85,B 0,C 180,E1 -4025.218,E2 -4025.218} C_VEL
LIN {X 0,Y 539.465,Z 590.941,A -85,B 0,C 180,E1 -4026.385,E2 -4026.385} C_VEL
LIN {X 0,Y 539.344,Z 603.204,A -85,B 0,C 180,E1 -4028.2,E2 -4028.2} C_VEL
LIN {X 0,Y 538.92,Z 623.553,A -85,B 0,C 180,E1 -4031.17,E2 -4031.17} C_VEL
LIN {X 0,Y 538.52,Z 642.3,A -85,B 0,C 180,E1 -4033.9,E2 -4033.9} C_VEL
LIN {X 0,Y 538.394,Z 651.544,A -85,B 0,C 180,E1 -4035.245,E2 -4035.245} C_VEL
LIN {X 0,Y 539.695,Z 660.585,A -85,B 0,C 180,E1 -4035.403,E2 -4035.403} C_VEL
LIN {X 0,Y 539.324,Z 759.962,A -85,B 0,C 180,E1 -4036.746,E2 -4036.746} C_VEL
LIN {X 0,Y 539.152,Z 773.228,A -85,B 0,C 180,E1 -4037.078,E2 -4037.078} C_VEL
LIN {X 0,Y 538.942,Z 786.495,A -85,B 0,C 180,E1 -4037.575,E2 -4037.575} C_VEL
LIN {X 0,Y 538.745,Z 798.37,A -85,B 0,C 180,E1 -4038.189,E2 -4038.189} C_VEL
LIN {X 0,Y 538.467,Z 810.49,A -85,B 0,C 180,E1 -4038.996,E2 -4038.996} C_VEL
LIN {X 0,Y 538.226,Z 820.649,A -85,B 0,C 180,E1 -4039.847,E2 -4039.847} C_VEL
LIN {X 0,Y 538.027,Z 829.788,A -85,B 0,C 180,E1 -4040.792,E2 -4040.792} C_VEL
LIN {X 0,Y 537.851,Z 838.69,A -85,B 0,C 180,E1 -4041.925,E2 -4041.925} C_VEL
LIN {X 0,Y 537.729,Z 845.85,A -85,B 0,C 180,E1 -4043.056,E2 -4043.056} C_VEL
LIN {X 0,Y 537.676,Z 852.367,A -85,B 0,C 180,E1 -4044.374,E2 -4044.374} C_VEL
LIN {X 0,Y 537.558,Z 856.677,A -85,B 0,C 180,E1 -4045.501,E2 -4045.501} C_VEL
LIN {X 0,Y 537.591,Z 858.958,A -85,B 0,C 180,E1 -4046.252,E2 -4046.252} C_VEL
LIN {X 0,Y 537.551,Z 860.807,A -85,B 0,C 180,E1 -4047.002,E2 -4047.002} C_VEL
LIN {X 0,Y 537.451,Z 863.183,A -85,B 0,C 180,E1 -4048.501,E2 -4048.501} C_VEL
LIN {X 0,Y 537.442,Z 864,A -85,B 0,C 180,E1 -4050,E2 -4050} C_VEL
LIN {X 0,Y 537.451,Z 863.185,A -85,B 0,C 180,E1 -4051.499,E2 -4051.499} C_VEL
LIN {X 0,Y 537.551,Z 860.81,A -85,B 0,C 180,E1 -4052.998,E2 -4052.998} C_VEL
LIN {X 0,Y 537.604,Z 857.896,A -85,B 0,C 180,E1 -4054.123,E2 -4054.123} C_VEL
LIN {X 0,Y 537.588,Z 853.949,A -85,B 0,C 180,E1 -4055.25,E2 -4055.25} C_VEL
LIN {X 0,Y 537.65,Z 849.083,A -85,B 0,C 180,E1 -4056.335,E2 -4056.335} C_VEL
LIN {X 0,Y 537.791,Z 842.468,A -85,B 0,C 180,E1 -4057.509,E2 -4057.509} C_VEL
LIN {X 0,Y 537.972,Z 834.479,A -85,B 0,C 180,E1 -4058.64,E2 -4058.64} C_VEL
LIN {X 0,Y 538.142,Z 826.336,A -85,B 0,C 180,E1 -4059.585,E2 -4059.585} C_VEL
LIN {X 0,Y 538.374,Z 816.401,A -85,B 0,C 180,E1 -4060.53,E2 -4060.53} C_VEL
LIN {X 0,Y 538.576,Z 806.595,A -85,B 0,C 180,E1 -4061.288,E2 -4061.288} C_VEL
LIN {X 0,Y 538.754,Z 795.551,A -85,B 0,C 180,E1 -4061.973,E2 -4061.973} C_VEL
LIN {X 0,Y 539.019,Z 783.111,A -85,B 0,C 180,E1 -4062.567,E2 -4062.567} C_VEL
LIN {X 0,Y 539.177,Z 770.099,A -85,B 0,C 180,E1 -4063.018,E2 -4063.018} C_VEL
LIN {X 0,Y 539.367,Z 757.125,A -85,B 0,C 180,E1 -4063.3,E2 -4063.3} C_VEL
LIN {X 0,Y 539.587,Z 658.94,A -85,B 0,C 180,E1 -4064.622,E2 -4064.622} C_VEL
LIN {X 0,Y 538.414,Z 651.503,A -85,B 0,C 180,E1 -4064.761,E2 -4064.761} C_VEL
LIN {X 0,Y 538.855,Z 628.652,A -85,B 0,C 180,E1 -4068.09,E2 -4068.09} C_VEL
LIN {X 0,Y 539.229,Z 608.701,A -85,B 0,C 180,E1 -4071.003,E2 -4071.003} C_VEL
LIN {X 0,Y 539.56,Z 592.447,A -85,B 0,C 180,E1 -4073.407,E2 -4073.407} C_VEL
LIN {X 0,Y 538.694,Z 586.518,A -85,B 0,C 180,E1 -4074.338,E2 -4074.338} C_VEL
LIN {X 0,Y 538.061,Z 583.463,A -85,B 0,C 180,E1 -4074.861,E2 -4074.861} C_VEL
LIN {X 0,Y 538.045,Z 583.466,A -85,B 0,C 180,E1 -4078.049,E2 -4078.049} C_VEL
LIN {X 0,Y 538.02,Z 583.468,A -85,B 0,C 180,E1 -4080.626,E2 -4080.626} C_VEL
LIN {X 0,Y 538.044,Z 583.458,A -85,B 0,C 180,E1 -4083.282,E2 -4083.282} C_VEL
LIN {X 0,Y 538.028,Z 583.463,A -85,B 0,C 180,E1 -4086.001,E2 -4086.001} C_VEL
LIN {X 0,Y 538.013,Z 583.467,A -85,B 0,C 180,E1 -4088.829,E2 -4088.829} C_VEL
LIN {X 0,Y 538.075,Z 583.461,A -85,B 0,C 180,E1 -4090.772,E2 -4090.772} C_VEL
LIN {X 0,Y 538.026,Z 583.462,A -85,B 0,C 180,E1 -4094.074,E2 -4094.074} C_VEL
LIN {X 0,Y 538.02,Z 583.463,A -85,B 0,C 180,E1 -4097.214,E2 -4097.214} C_VEL
LIN {X 0,Y 538.025,Z 583.462,A -85,B 0,C 180,E1 -4100.203,E2 -4100.203} C_VEL
LIN {X 0,Y 538.025,Z 583.466,A -85,B 0,C 180,E1 -4103.067,E2 -4103.067} C_VEL
LIN {X 0,Y 538.021,Z 583.461,A -85,B 0,C 180,E1 -4105.826,E2 -4105.826} C_VEL
LIN {X 0,Y 538.018,Z 583.465,A -85,B 0,C 180,E1 -4108.499,E2 -4108.499} C_VEL
LIN {X 0,Y 538.052,Z 583.464,A -85,B 0,C 180,E1 -4111.099,E2 -4111.099} C_VEL
LIN {X 0,Y 538.043,Z 583.459,A -85,B 0,C 180,E1 -4113.633,E2 -4113.633} C_VEL
LIN {X 0,Y 538.015,Z 583.462,A -85,B 0,C 180,E1 -4116.117,E2 -4116.117} C_VEL
LIN {X 0,Y 538.034,Z 583.465,A -85,B 0,C 180,E1 -4119.348,E2 -4119.348} C_VEL
LIN {X 0,Y 538.064,Z 583.457,A -85,B 0,C 180,E1 -4122.517,E2 -4122.517} C_VEL
LIN {X 0,Y 538.054,Z 583.46,A -85,B 0,C 180,E1 -4125.63,E2 -4125.63} C_VEL
LIN {X 0,Y 538.08,Z 583.455,A -85,B 0,C 180,E1 -4128.701,E2 -4128.701} C_VEL
LIN {X 0,Y 538.082,Z 583.456,A -85,B 0,C 180,E1 -4131.739,E2 -4131.739} C_VEL
LIN {X 0,Y 538.178,Z 583.443,A -85,B 0,C 180,E1 -4134.755,E2 -4134.755} C_VEL
LIN {X 0,Y 538.158,Z 583.448,A -85,B 0,C 180,E1 -4137.754,E2 -4137.754} C_VEL
LIN {X 0,Y 538.176,Z 583.442,A -85,B 0,C 180,E1 -4140.748,E2 -4140.748} C_VEL
LIN {X 0,Y 538.135,Z 583.449,A -85,B 0,C 180,E1 -4142.994,E2 -4142.994} C_VEL
LIN {X 0,Y 538.114,Z 583.452,A -85,B 0,C 180,E1 -4145.997,E2 -4145.997} C_VEL
LIN {X 0,Y 538.067,Z 583.457,A -85,B 0,C 180,E1 -4149.017,E2 -4149.017} C_VEL
LIN {X 0,Y 538.073,Z 583.458,A -85,B 0,C 180,E1 -4152.062,E2 -4152.062} C_VEL
LIN {X 0,Y 538.034,Z 583.461,A -85,B 0,C 180,E1 -4155.144,E2 -4155.144} C_VEL
LIN {X 0,Y 538.024,Z 583.463,A -85,B 0,C 180,E1 -4158.27,E2 -4158.27} C_VEL
LIN {X 0,Y 538.031,Z 583.46,A -85,B 0,C 180,E1 -4160.651,E2 -4160.651} C_VEL
LIN {X 0,Y 538.013,Z 583.472,A -85,B 0,C 180,E1 -4163.887,E2 -4163.887} C_VEL
LIN {X 0,Y 538.04,Z 583.462,A -85,B 0,C 180,E1 -4166.366,E2 -4166.366} C_VEL
LIN {X 0,Y 538.046,Z 583.458,A -85,B 0,C 180,E1 -4168.939,E2 -4168.939} C_VEL
LIN {X 0,Y 538.018,Z 583.469,A -85,B 0,C 180,E1 -4171.891,E2 -4171.891} C_VEL
LIN {X 0,Y 538.021,Z 583.463,A -85,B 0,C 180,E1 -4174.621,E2 -4174.621} C_VEL
LIN {X 0,Y 538.001,Z 583.463,A -85,B 0,C 180,E1 -4177.171,E2 -4177.171} C_VEL
LIN {X 0,Y 538.04,Z 583.459,A -85,B 0,C 180,E1 -4180.275,E2 -4180.275} C_VEL
LIN {X 0,Y 537.39,Z 583.542,A -85,B 0,C 180,E1 -4180.9,E2 -4180.9} C_VEL
LIN {X 0,Y 534.53,Z 583.901,A -85,B 0,C 180,E1 -4181.915,E2 -4181.915} C_VEL
LIN {X 0,Y 532.097,Z 584.201,A -85,B 0,C 180,E1 -4182.732,E2 -4182.732} C_VEL
LIN {X 0,Y 531.045,Z 584.33,A -85,B 0,C 180,E1 -4183.363,E2 -4183.363} C_VEL
LIN {X 0,Y 530.956,Z 584.341,A -85,B 0,C 180,E1 -4183.576,E2 -4183.576} C_VEL
LIN {X 0,Y 530.958,Z 584.347,A -85,B 0,C 180,E1 -4186.506,E2 -4186.506} C_VEL
LIN {X 0,Y 530.981,Z 584.339,A -85,B 0,C 180,E1 -4188.976,E2 -4188.976} C_VEL
LIN {X 0,Y 530.952,Z 584.341,A -85,B 0,C 180,E1 -4191.53,E2 -4191.53} C_VEL
LIN {X 0,Y 530.976,Z 584.348,A -85,B 0,C 180,E1 -4194.383,E2 -4194.383} C_VEL
LIN {X 0,Y 530.969,Z 584.34,A -85,B 0,C 180,E1 -4197.134,E2 -4197.134} C_VEL
LIN {X 0,Y 530.964,Z 584.341,A -85,B 0,C 180,E1 -4199.804,E2 -4199.804} C_VEL
LIN {X 0,Y 531.011,Z 584.342,A -85,B 0,C 180,E1 -4202.467,E2 -4202.467} C_VEL
LIN {X 0,Y 531.001,Z 584.34,A -85,B 0,C 180,E1 -4204.943,E2 -4204.943} C_VEL
LIN {X 0,Y 530.967,Z 584.343,A -85,B 0,C 180,E1 -4208.247,E2 -4208.247} C_VEL
LIN {X 0,Y 530.994,Z 584.345,A -85,B 0,C 180,E1 -4210.678,E2 -4210.678} C_VEL
LIN {X 0,Y 530.989,Z 584.342,A -85,B 0,C 180,E1 -4213.072,E2 -4213.072} C_VEL
LIN {X 0,Y 531.016,Z 584.335,A -85,B 0,C 180,E1 -4215.436,E2 -4215.436} C_VEL
LIN {X 0,Y 531.034,Z 584.336,A -85,B 0,C 180,E1 -4218.55,E2 -4218.55} C_VEL
LIN {X 0,Y 531.054,Z 584.329,A -85,B 0,C 180,E1 -4221.63,E2 -4221.63} C_VEL
LIN {X 0,Y 531.119,Z 584.326,A -85,B 0,C 180,E1 -4224.685,E2 -4224.685} C_VEL
LIN {X 0,Y 531.139,Z 584.319,A -85,B 0,C 180,E1 -4227.725,E2 -4227.725} C_VEL
LIN {X 0,Y 531.15,Z 584.321,A -85,B 0,C 180,E1 -4230.758,E2 -4230.758} C_VEL
LIN {X 0,Y 531.104,Z 584.331,A -85,B 0,C 180,E1 -4233.034,E2 -4233.034} C_VEL
LIN {X 0,Y 531.073,Z 584.326,A -85,B 0,C 180,E1 -4236.077,E2 -4236.077} C_VEL
LIN {X 0,Y 531.053,Z 584.329,A -85,B 0,C 180,E1 -4238.37,E2 -4238.37} C_VEL
LIN {X 0,Y 531.048,Z 584.333,A -85,B 0,C 180,E1 -4241.672,E2 -4241.672} C_VEL
LIN {X 0,Y 531.027,Z 584.336,A -85,B 0,C 180,E1 -4244.956,E2 -4244.956} C_VEL
LIN {X 0,Y 531.013,Z 584.339,A -85,B 0,C 180,E1 -4247.722,E2 -4247.722} C_VEL
LIN {X 0,Y 530.996,Z 584.34,A -85,B 0,C 180,E1 -4250.938,E2 -4250.938} C_VEL
LIN {X 0,Y 530.967,Z 584.344,A -85,B 0,C 180,E1 -4254.224,E2 -4254.224} C_VEL
LIN {X 0,Y 531.055,Z 584.372,A -85,B 0,C 180,E1 -4256.105,E2 -4256.105} C_VEL
LIN {X 0,Y 531.431,Z 588.295,A -85,B 0,C 180,E1 -4256.932,E2 -4256.932} C_VEL
LIN {X 0,Y 531.129,Z 603.103,A -85,B 0,C 180,E1 -4259.967,E2 -4259.967} C_VEL
LIN {X 0,Y 531.112,Z 603.783,A -85,B 0,C 180,E1 -4260.105,E2 -4260.105} C_VEL
LIN {X 0,Y 532.773,Z 614.112,A -85,B 0,C 180,E1 -4260.302,E2 -4260.302} C_VEL
LIN {X 0,Y 532.395,Z 710.96,A -85,B 0,C 180,E1 -4261.635,E2 -4261.635} C_VEL
LIN {X 0,Y 532.2,Z 724.581,A -85,B 0,C 180,E1 -4261.995,E2 -4261.995} C_VEL
LIN {X 0,Y 532.003,Z 737.566,A -85,B 0,C 180,E1 -4262.505,E2 -4262.505} C_VEL
LIN {X 0,Y 531.729,Z 749.613,A -85,B 0,C 180,E1 -4263.151,E2 -4263.151} C_VEL
LIN {X 0,Y 531.425,Z 761.463,A -85,B 0,C 180,E1 -4263.968,E2 -4263.968} C_VEL
LIN {X 0,Y 531.19,Z 771.971,A -85,B 0,C 180,E1 -4264.886,E2 -4264.886} C_VEL
LIN {X 0,Y 530.952,Z 781.22,A -85,B 0,C 180,E1 -4265.883,E2 -4265.883} C_VEL
LIN {X 0,Y 530.77,Z 789.482,A -85,B 0,C 180,E1 -4266.976,E2 -4266.976} C_VEL
LIN {X 0,Y 530.663,Z 795.862,A -85,B 0,C 180,E1 -4268.012,E2 -4268.012} C_VEL
LIN {X 0,Y 530.561,Z 801.963,A -85,B 0,C 180,E1 -4269.247,E2 -4269.247} C_VEL
LIN {X 0,Y 530.453,Z 806.661,A -85,B 0,C 180,E1 -4270.48,E2 -4270.48} C_VEL
LIN {X 0,Y 530.48,Z 809.591,A -85,B 0,C 180,E1 -4271.483,E2 -4271.483} C_VEL
LIN {X 0,Y 530.411,Z 811.776,A -85,B 0,C 180,E1 -4272.511,E2 -4272.511} C_VEL
LIN {X 0,Y 530.349,Z 813.215,A -85,B 0,C 180,E1 -4273.556,E2 -4273.556} C_VEL
LIN {X 0,Y 530.375,Z 813.916,A -85,B 0,C 180,E1 -4274.611,E2 -4274.611} C_VEL
LIN {X 0,Y 530.376,Z 813.857,A -85,B 0,C 180,E1 -4275.687,E2 -4275.687} C_VEL
LIN {X 0,Y 530.356,Z 812.948,A -85,B 0,C 180,E1 -4276.787,E2 -4276.787} C_VEL
LIN {X 0,Y 530.435,Z 811.168,A -85,B 0,C 180,E1 -4277.898,E2 -4277.898} C_VEL
LIN {X 0,Y 530.44,Z 808.403,A -85,B 0,C 180,E1 -4279.042,E2 -4279.042} C_VEL
LIN {X 0,Y 530.511,Z 804.553,A -85,B 0,C 180,E1 -4280.205,E2 -4280.205} C_VEL
LIN {X 0,Y 530.617,Z 798.911,A -85,B 0,C 180,E1 -4281.501,E2 -4281.501} C_VEL
LIN {X 0,Y 530.752,Z 791.404,A -85,B 0,C 180,E1 -4282.82,E2 -4282.82} C_VEL
LIN {X 0,Y 530.921,Z 783.036,A -85,B 0,C 180,E1 -4283.989,E2 -4283.989} C_VEL
LIN {X 0,Y 531.148,Z 774.188,A -85,B 0,C 180,E1 -4284.984,E2 -4284.984} C_VEL
LIN {X 0,Y 531.373,Z 764.036,A -85,B 0,C 180,E1 -4285.913,E2 -4285.913} C_VEL
LIN {X 0,Y 531.666,Z 752.943,A -85,B 0,C 180,E1 -4286.731,E2 -4286.731} C_VEL
LIN {X 0,Y 531.869,Z 741.085,A -85,B 0,C 180,E1 -4287.414,E2 -4287.414} C_VEL
LIN {X 0,Y 532.145,Z 728.258,A -85,B 0,C 180,E1 -4287.969,E2 -4287.969} C_VEL
LIN {X 0,Y 532.341,Z 715.839,A -85,B 0,C 180,E1 -4288.347,E2 -4288.347} C_VEL
LIN {X 0,Y 532.467,Z 701.531,A -85,B 0,C 180,E1 -4288.605,E2 -4288.605} C_VEL
LIN {X 0,Y 532.669,Z 612.694,A -85,B 0,C 180,E1 -4289.81,E2 -4289.81} C_VEL
LIN {X 0,Y 531.123,Z 603.883,A -85,B 0,C 180,E1 -4289.978,E2 -4289.978} C_VEL
LIN {X 0,Y 531.441,Z 588.91,A -85,B 0,C 180,E1 -4293.068,E2 -4293.068} C_VEL
LIN {X 0,Y 531.052,Z 584.338,A -85,B 0,C 180,E1 -4294.053,E2 -4294.053} C_VEL
LIN {X 0,Y 530.955,Z 584.351,A -85,B 0,C 180,E1 -4296.604,E2 -4296.604} C_VEL
LIN {X 0,Y 531.014,Z 584.336,A -85,B 0,C 180,E1 -4299.873,E2 -4299.873} C_VEL
LIN {X 0,Y 530.982,Z 584.342,A -85,B 0,C 180,E1 -4303.071,E2 -4303.071} C_VEL
LIN {X 0,Y 531.008,Z 584.336,A -85,B 0,C 180,E1 -4305.436,E2 -4305.436} C_VEL
LIN {X 0,Y 531.036,Z 584.339,A -85,B 0,C 180,E1 -4308.55,E2 -4308.55} C_VEL
LIN {X 0,Y 531.052,Z 584.331,A -85,B 0,C 180,E1 -4311.63,E2 -4311.63} C_VEL
LIN {X 0,Y 531.136,Z 584.327,A -85,B 0,C 180,E1 -4314.686,E2 -4314.686} C_VEL
LIN {X 0,Y 531.131,Z 584.32,A -85,B 0,C 180,E1 -4317.725,E2 -4317.725} C_VEL
LIN {X 0,Y 531.147,Z 584.326,A -85,B 0,C 180,E1 -4320.759,E2 -4320.759} C_VEL
LIN {X 0,Y 531.102,Z 584.33,A -85,B 0,C 180,E1 -4323.035,E2 -4323.035} C_VEL
LIN {X 0,Y 531.082,Z 584.326,A -85,B 0,C 180,E1 -4326.077,E2 -4326.077} C_VEL
LIN {X 0,Y 531.029,Z 584.339,A -85,B 0,C 180,E1 -4329.139,E2 -4329.139} C_VEL
LIN {X 0,Y 531.052,Z 584.331,A -85,B 0,C 180,E1 -4331.678,E2 -4331.678} C_VEL
LIN {X 0,Y 531.021,Z 584.341,A -85,B 0,C 180,E1 -4334.956,E2 -4334.956} C_VEL
LIN {X 0,Y 531.008,Z 584.337,A -85,B 0,C 180,E1 -4337.723,E2 -4337.723} C_VEL
LIN {X 0,Y 530.994,Z 584.343,A -85,B 0,C 180,E1 -4340.939,E2 -4340.939} C_VEL
LIN {X 0,Y 530.972,Z 584.339,A -85,B 0,C 180,E1 -4344.225,E2 -4344.225} C_VEL
LIN {X 0,Y 531.005,Z 584.336,A -85,B 0,C 180,E1 -4346.744,E2 -4346.744} C_VEL
LIN {X 0,Y 530.993,Z 584.344,A -85,B 0,C 180,E1 -4349.322,E2 -4349.322} C_VEL
LIN {X 0,Y 530.974,Z 584.337,A -85,B 0,C 180,E1 -4352.104,E2 -4352.104} C_VEL
LIN {X 0,Y 530.985,Z 584.34,A -85,B 0,C 180,E1 -4354.855,E2 -4354.855} C_VEL
LIN {X 0,Y 530.968,Z 584.346,A -85,B 0,C 180,E1 -4357.508,E2 -4357.508} C_VEL
LIN {X 0,Y 530.981,Z 584.338,A -85,B 0,C 180,E1 -4360.433,E2 -4360.433} C_VEL
LIN {X 0,Y 530.963,Z 584.349,A -85,B 0,C 180,E1 -4363.495,E2 -4363.495} C_VEL
LIN {X 0,Y 530.961,Z 584.341,A -85,B 0,C 180,E1 -4366.506,E2 -4366.506} C_VEL
LIN {X 0,Y 531.024,Z 584.342,A -85,B 0,C 180,E1 -4369.572,E2 -4369.572} C_VEL
LIN {X 0,Y 530.968,Z 584.341,A -85,B 0,C 180,E1 -4372.578,E2 -4372.578} C_VEL
LIN {X 0,Y 531.001,Z 584.342,A -85,B 0,C 180,E1 -4375.312,E2 -4375.312} C_VEL
LIN {X 0,Y 530.971,Z 584.344,A -85,B 0,C 180,E1 -4378.033,E2 -4378.033} C_VEL
LIN {X 0,Y 530.989,Z 584.34,A -85,B 0,C 180,E1 -4380.875,E2 -4380.875} C_VEL
LIN {X 0,Y 531.002,Z 584.341,A -85,B 0,C 180,E1 -4383.257,E2 -4383.257} C_VEL
LIN {X 0,Y 531.057,Z 584.504,A -85,B 0,C 180,E1 -4385.061,E2 -4385.061} C_VEL
LIN {X 0,Y 532.575,Z 593.311,A -85,B 0,C 180,E1 -4386.473,E2 -4386.473} C_VEL
LIN {X 0,Y 532.204,Z 611.003,A -85,B 0,C 180,E1 -4389.112,E2 -4389.112} C_VEL
LIN {X 0,Y 531.764,Z 631.301,A -85,B 0,C 180,E1 -4392.098,E2 -4392.098} C_VEL
LIN {X 0,Y 531.403,Z 651.482,A -85,B 0,C 180,E1 -4395.037,E2 -4395.037} C_VEL
LIN {X 0,Y 532.845,Z 661.103,A -85,B 0,C 180,E1 -4395.219,E2 -4395.219} C_VEL
LIN {X 0,Y 532.44,Z 759.962,A -85,B 0,C 180,E1 -4396.572,E2 -4396.572} C_VEL
LIN {X 0,Y 532.23,Z 773.227,A -85,B 0,C 180,E1 -4396.907,E2 -4396.907} C_VEL
LIN {X 0,Y 532.012,Z 786.495,A -85,B 0,C 180,E1 -4397.411,E2 -4397.411} C_VEL
LIN {X 0,Y 531.805,Z 797.935,A -85,B 0,C 180,E1 -4398.006,E2 -4398.006} C_VEL
LIN {X 0,Y 531.526,Z 809.197,A -85,B 0,C 180,E1 -4398.754,E2 -4398.754} C_VEL
LIN {X 0,Y 531.256,Z 819.608,A -85,B 0,C 180,E1 -4399.616,E2 -4399.616} C_VEL
LIN {X 0,Y 531.06,Z 828.115,A -85,B 0,C 180,E1 -4400.478,E2 -4400.478} C_VEL
LIN {X 0,Y 530.887,Z 835.962,A -85,B 0,C 180,E1 -4401.435,E2 -4401.435} C_VEL
LIN {X 0,Y 530.685,Z 843.623,A -85,B 0,C 180,E1 -4402.581,E2 -4402.581} C_VEL
LIN {X 0,Y 530.604,Z 850.68,A -85,B 0,C 180,E1 -4403.918,E2 -4403.918} C_VEL
LIN {X 0,Y 530.459,Z 855.373,A -85,B 0,C 180,E1 -4405.06,E2 -4405.06} C_VEL
LIN {X 0,Y 530.516,Z 858.958,A -85,B 0,C 180,E1 -4406.202,E2 -4406.202} C_VEL
LIN {X 0,Y 530.457,Z 860.807,A -85,B 0,C 180,E1 -4406.962,E2 -4406.962} C_VEL
LIN {X 0,Y 530.41,Z 862.194,A -85,B 0,C 180,E1 -4407.722,E2 -4407.722} C_VEL
LIN {X 0,Y 530.344,Z 863.786,A -85,B 0,C 180,E1 -4409.241,E2 -4409.241} C_VEL
LIN {X 0,Y 530.342,Z 864,A -85,B 0,C 180,E1 -4410,E2 -4410} C_VEL
LIN {X 0,Y 530.361,Z 863.184,A -85,B 0,C 180,E1 -4411.519,E2 -4411.519} C_VEL
LIN {X 0,Y 530.41,Z 862.197,A -85,B 0,C 180,E1 -4412.278,E2 -4412.278} C_VEL
LIN {X 0,Y 530.457,Z 860.81,A -85,B 0,C 180,E1 -4413.038,E2 -4413.038} C_VEL
LIN {X 0,Y 530.523,Z 857.896,A -85,B 0,C 180,E1 -4414.178,E2 -4414.178} C_VEL
LIN {X 0,Y 530.525,Z 853.949,A -85,B 0,C 180,E1 -4415.321,E2 -4415.321} C_VEL
LIN {X 0,Y 530.599,Z 848.265,A -85,B 0,C 180,E1 -4416.582,E2 -4416.582} C_VEL
LIN {X 0,Y 530.758,Z 841.237,A -85,B 0,C 180,E1 -4417.8,E2 -4417.8} C_VEL
LIN {X 0,Y 530.93,Z 832.994,A -85,B 0,C 180,E1 -4418.948,E2 -4418.948} C_VEL
LIN {X 0,Y 531.137,Z 824.542,A -85,B 0,C 180,E1 -4419.905,E2 -4419.905} C_VEL
LIN {X 0,Y 531.408,Z 814.095,A -85,B 0,C 180,E1 -4420.863,E2 -4420.863} C_VEL
LIN {X 0,Y 531.693,Z 803.362,A -85,B 0,C 180,E1 -4421.655,E2 -4421.655} C_VEL
LIN {X 0,Y 531.932,Z 792.41,A -85,B 0,C 180,E1 -4422.301,E2 -4422.301} C_VEL
LIN {X 0,Y 532.132,Z 780.772,A -85,B 0,C 180,E1 -4422.829,E2 -4422.829} C_VEL
LIN {X 0,Y 532.322,Z 767.357,A -85,B 0,C 180,E1 -4423.261,E2 -4423.261} C_VEL
LIN {X 0,Y 532.479,Z 754.107,A -85,B 0,C 180,E1 -4423.524,E2 -4423.524} C_VEL
LIN {X 0,Y 532.659,Z 659.403,A -85,B 0,C 180,E1 -4424.81,E2 -4424.81} C_VEL
LIN {X 0,Y 531.411,Z 651.459,A -85,B 0,C 180,E1 -4424.966,E2 -4424.966} C_VEL
LIN {X 0,Y 531.86,Z 629.751,A -85,B 0,C 180,E1 -4428.135,E2 -4428.135} C_VEL
LIN {X 0,Y 532.269,Z 609.785,A -85,B 0,C 180,E1 -4431.088,E2 -4431.088} C_VEL
LIN {X 0,Y 532.62,Z 593.531,A -85,B 0,C 180,E1 -4433.525,E2 -4433.525} C_VEL
LIN {X 0,Y 531.244,Z 585.406,A -85,B 0,C 180,E1 -4434.836,E2 -4434.836} C_VEL
LIN {X 0,Y 531.06,Z 584.334,A -85,B 0,C 180,E1 -4435.054,E2 -4435.054} C_VEL
LIN {X 0,Y 531.016,Z 584.338,A -85,B 0,C 180,E1 -4437.595,E2 -4437.595} C_VEL
LIN {X 0,Y 530.974,Z 584.346,A -85,B 0,C 180,E1 -4440.644,E2 -4440.644} C_VEL
LIN {X 0,Y 530.99,Z 584.338,A -85,B 0,C 180,E1 -4443.772,E2 -4443.772} C_VEL
LIN {X 0,Y 530.97,Z 584.348,A -85,B 0,C 180,E1 -4446.556,E2 -4446.556} C_VEL
LIN {X 0,Y 531.003,Z 584.336,A -85,B 0,C 180,E1 -4449.856,E2 -4449.856} C_VEL
LIN {X 0,Y 530.977,Z 584.346,A -85,B 0,C 180,E1 -4452.456,E2 -4452.456} C_VEL
LIN {X 0,Y 530.984,Z 584.337,A -85,B 0,C 180,E1 -4455.62,E2 -4455.62} C_VEL
LIN {X 0,Y 530.996,Z 584.343,A -85,B 0,C 180,E1 -4458.564,E2 -4458.564} C_VEL
LIN {X 0,Y 530.955,Z 584.341,A -85,B 0,C 180,E1 -4461.529,E2 -4461.529} C_VEL
LIN {X 0,Y 530.976,Z 584.342,A -85,B 0,C 180,E1 -4464.381,E2 -4464.381} C_VEL
LIN {X 0,Y 530.966,Z 584.345,A -85,B 0,C 180,E1 -4467.133,E2 -4467.133} C_VEL
LIN {X 0,Y 530.979,Z 584.338,A -85,B 0,C 180,E1 -4469.803,E2 -4469.803} C_VEL
LIN {X 0,Y 531.011,Z 584.337,A -85,B 0,C 180,E1 -4472.465,E2 -4472.465} C_VEL
LIN {X 0,Y 531,Z 584.344,A -85,B 0,C 180,E1 -4474.942,E2 -4474.942} C_VEL
LIN {X 0,Y 530.963,Z 584.34,A -85,B 0,C 180,E1 -4478.246,E2 -4478.246} C_VEL
LIN {X 0,Y 530.989,Z 584.34,A -85,B 0,C 180,E1 -4480.677,E2 -4480.677} C_VEL
LIN {X 0,Y 530.983,Z 584.346,A -85,B 0,C 180,E1 -4483.071,E2 -4483.071} C_VEL
LIN {X 0,Y 531.009,Z 584.34,A -85,B 0,C 180,E1 -4485.435,E2 -4485.435} C_VEL
LIN {X 0,Y 531.037,Z 584.332,A -85,B 0,C 180,E1 -4488.549,E2 -4488.549} C_VEL
LIN {X 0,Y 531.051,Z 584.334,A -85,B 0,C 180,E1 -4491.629,E2 -4491.629} C_VEL
LIN {X 0,Y 531.134,Z 584.32,A -85,B 0,C 180,E1 -4494.685,E2 -4494.685} C_VEL
LIN {X 0,Y 531.13,Z 584.324,A -85,B 0,C 180,E1 -4497.725,E2 -4497.725} C_VEL
LIN {X 0,Y 531.146,Z 584.318,A -85,B 0,C 180,E1 -4500.758,E2 -4500.758} C_VEL
LIN {X 0,Y 531.101,Z 584.326,A -85,B 0,C 180,E1 -4503.034,E2 -4503.034} C_VEL
LIN {X 0,Y 531.074,Z 584.329,A -85,B 0,C 180,E1 -4506.077,E2 -4506.077} C_VEL
LIN {X 0,Y 531.026,Z 584.335,A -85,B 0,C 180,E1 -4509.138,E2 -4509.138} C_VEL
LIN {X 0,Y 531.03,Z 584.334,A -85,B 0,C 180,E1 -4512.225,E2 -4512.225} C_VEL
LIN {X 0,Y 530.985,Z 584.341,A -85,B 0,C 180,E1 -4515.35,E2 -4515.35} C_VEL
LIN {X 0,Y 531.005,Z 584.344,A -85,B 0,C 180,E1 -4517.722,E2 -4517.722} C_VEL
LIN {X 0,Y 530.991,Z 584.336,A -85,B 0,C 180,E1 -4520.938,E2 -4520.938} C_VEL
LIN {X 0,Y 530.969,Z 584.344,A -85,B 0,C 180,E1 -4524.225,E2 -4524.225} C_VEL
LIN {X 0,Y 531.002,Z 584.335,A -85,B 0,C 180,E1 -4526.743,E2 -4526.743} C_VEL
LIN {X 0,Y 530.99,Z 584.338,A -85,B 0,C 180,E1 -4529.322,E2 -4529.322} C_VEL
LIN {X 0,Y 530.97,Z 584.348,A -85,B 0,C 180,E1 -4532.103,E2 -4532.103} C_VEL
LIN {X 0,Y 530.978,Z 584.339,A -85,B 0,C 180,E1 -4534.854,E2 -4534.854} C_VEL
LIN {X 0,Y 530.958,Z 584.342,A -85,B 0,C 180,E1 -4537.508,E2 -4537.508} C_VEL
LIN {X 0,Y 531.019,Z 584.339,A -85,B 0,C 180,E1 -4540.429,E2 -4540.429} C_VEL
LIN {X 0,Y 530.959,Z 584.341,A -85,B 0,C 180,E1 -4543.495,E2 -4543.495} C_VEL
LIN {X 0,Y 530.956,Z 584.341,A -85,B 0,C 180,E1 -4543.576,E2 -4543.576} C_VEL
LIN {X 0,Y 530.283,Z 584.434,A -85,B 0,C 180,E1 -4544.21,E2 -4544.21} C_VEL
LIN {X 0,Y 527.435,Z 584.785,A -85,B 0,C 180,E1 -4545.239,E2 -4545.239} C_VEL
LIN {X 0,Y 525.031,Z 585.085,A -85,B 0,C 180,E1 -4546.067,E2 -4546.067} C_VEL
LIN {X 0,Y 523.999,Z 585.212,A -85,B 0,C 180,E1 -4546.707,E2 -4546.707} C_VEL
LIN {X 0,Y 523.914,Z 585.219,A -85,B 0,C 180,E1 -4546.923,E2 -4546.923} C_VEL
LIN {X 0,Y 523.94,Z 585.218,A -85,B 0,C 180,E1 -4549.921,E2 -4549.921} C_VEL
LIN {X 0,Y 523.905,Z 585.222,A -85,B 0,C 180,E1 -4552.869,E2 -4552.869} C_VEL
LIN {X 0,Y 523.94,Z 585.215,A -85,B 0,C 180,E1 -4555.711,E2 -4555.711} C_VEL
LIN {X 0,Y 523.926,Z 585.226,A -85,B 0,C 180,E1 -4558.457,E2 -4558.457} C_VEL
LIN {X 0,Y 523.935,Z 585.217,A -85,B 0,C 180,E1 -4561.126,E2 -4561.126} C_VEL
LIN {X 0,Y 523.979,Z 585.211,A -85,B 0,C 180,E1 -4563.981,E2 -4563.981} C_VEL
LIN {X 0,Y 523.932,Z 585.22,A -85,B 0,C 180,E1 -4566.271,E2 -4566.271} C_VEL
LIN {X 0,Y 523.942,Z 585.223,A -85,B 0,C 180,E1 -4568.767,E2 -4568.767} C_VEL
LIN {X 0,Y 523.95,Z 585.216,A -85,B 0,C 180,E1 -4571.221,E2 -4571.221} C_VEL
LIN {X 0,Y 523.937,Z 585.215,A -85,B 0,C 180,E1 -4573.639,E2 -4573.639} C_VEL
LIN {X 0,Y 523.937,Z 585.216,A -85,B 0,C 180,E1 -4576.028,E2 -4576.028} C_VEL
LIN {X 0,Y 524.009,Z 585.209,A -85,B 0,C 180,E1 -4578.394,E2 -4578.394} C_VEL
LIN {X 0,Y 524.002,Z 585.209,A -85,B 0,C 180,E1 -4581.516,E2 -4581.516} C_VEL
LIN {X 0,Y 524.079,Z 585.202,A -85,B 0,C 180,E1 -4584.614,E2 -4584.614} C_VEL
LIN {X 0,Y 524.111,Z 585.195,A -85,B 0,C 180,E1 -4587.695,E2 -4587.695} C_VEL
LIN {X 0,Y 524.12,Z 585.197,A -85,B 0,C 180,E1 -4590.768,E2 -4590.768} C_VEL
LIN {X 0,Y 524.071,Z 585.208,A -85,B 0,C 180,E1 -4593.075,E2 -4593.075} C_VEL
LIN {X 0,Y 524.034,Z 585.203,A -85,B 0,C 180,E1 -4596.159,E2 -4596.159} C_VEL
LIN {X 0,Y 524.001,Z 585.208,A -85,B 0,C 180,E1 -4598.484,E2 -4598.484} C_VEL
LIN {X 0,Y 524,Z 585.211,A -85,B 0,C 180,E1 -4601.739,E2 -4601.739} C_VEL
LIN {X 0,Y 523.989,Z 585.214,A -85,B 0,C 180,E1 -4605.052,E2 -4605.052} C_VEL
LIN {X 0,Y 523.961,Z 585.214,A -85,B 0,C 180,E1 -4607.969,E2 -4607.969} C_VEL
LIN {X 0,Y 523.968,Z 585.213,A -85,B 0,C 180,E1 -4610.41,E2 -4610.41} C_VEL
LIN {X 0,Y 523.913,Z 585.222,A -85,B 0,C 180,E1 -4612.893,E2 -4612.893} C_VEL
LIN {X 0,Y 524.007,Z 585.284,A -85,B 0,C 180,E1 -4615.988,E2 -4615.988} C_VEL
LIN {X 0,Y 524.452,Z 589.538,A -85,B 0,C 180,E1 -4616.889,E2 -4616.889} C_VEL
LIN {X 0,Y 524.132,Z 604.104,A -85,B 0,C 180,E1 -4619.909,E2 -4619.909} C_VEL
LIN {X 0,Y 525.886,Z 614.189,A -85,B 0,C 180,E1 -4620.103,E2 -4620.103} C_VEL
LIN {X 0,Y 525.485,Z 710.896,A -85,B 0,C 180,E1 -4621.453,E2 -4621.453} C_VEL
LIN {X 0,Y 525.285,Z 724.233,A -85,B 0,C 180,E1 -4621.804,E2 -4621.804} C_VEL
LIN {X 0,Y 525.078,Z 737.189,A -85,B 0,C 180,E1 -4622.312,E2 -4622.312} C_VEL
LIN {X 0,Y 524.789,Z 749.546,A -85,B 0,C 180,E1 -4622.978,E2 -4622.978} C_VEL
LIN {X 0,Y 524.51,Z 759.752,A -85,B 0,C 180,E1 -4623.679,E2 -4623.679} C_VEL
LIN {X 0,Y 524.202,Z 770.737,A -85,B 0,C 180,E1 -4624.618,E2 -4624.618} C_VEL
LIN {X 0,Y 523.997,Z 779.705,A -85,B 0,C 180,E1 -4625.573,E2 -4625.573} C_VEL
LIN {X 0,Y 523.776,Z 788.571,A -85,B 0,C 180,E1 -4626.736,E2 -4626.736} C_VEL
LIN {X 0,Y 523.596,Z 795.496,A -85,B 0,C 180,E1 -4627.852,E2 -4627.852} C_VEL
LIN {X 0,Y 523.466,Z 801.78,A -85,B 0,C 180,E1 -4629.124,E2 -4629.124} C_VEL
LIN {X 0,Y 523.411,Z 805.697,A -85,B 0,C 180,E1 -4630.128,E2 -4630.128} C_VEL
LIN {X 0,Y 523.378,Z 810.148,A -85,B 0,C 180,E1 -4631.677,E2 -4631.677} C_VEL
LIN {X 0,Y 523.318,Z 811.605,A -85,B 0,C 180,E1 -4632.386,E2 -4632.386} C_VEL
LIN {X 0,Y 523.25,Z 813.185,A -85,B 0,C 180,E1 -4633.507,E2 -4633.507} C_VEL
LIN {X 0,Y 523.275,Z 813.918,A -85,B 0,C 180,E1 -4634.616,E2 -4634.616} C_VEL
LIN {X 0,Y 523.275,Z 813.854,A -85,B 0,C 180,E1 -4635.702,E2 -4635.702} C_VEL
LIN {X 0,Y 523.258,Z 812.994,A -85,B 0,C 180,E1 -4636.766,E2 -4636.766} C_VEL
LIN {X 0,Y 523.353,Z 811.381,A -85,B 0,C 180,E1 -4637.822,E2 -4637.822} C_VEL
LIN {X 0,Y 523.379,Z 809.065,A -85,B 0,C 180,E1 -4638.855,E2 -4638.855} C_VEL
LIN {X 0,Y 523.414,Z 805.791,A -85,B 0,C 180,E1 -4639.937,E2 -4639.937} C_VEL
LIN {X 0,Y 523.478,Z 801.011,A -85,B 0,C 180,E1 -4641.138,E2 -4641.138} C_VEL
LIN {X 0,Y 523.584,Z 794.764,A -85,B 0,C 180,E1 -4642.366,E2 -4642.366} C_VEL
LIN {X 0,Y 523.789,Z 786.78,A -85,B 0,C 180,E1 -4643.614,E2 -4643.614} C_VEL
LIN {X 0,Y 524.047,Z 777.356,A -85,B 0,C 180,E1 -4644.784,E2 -4644.784} C_VEL
LIN {X 0,Y 524.309,Z 767.855,A -85,B 0,C 180,E1 -4645.738,E2 -4645.738} C_VEL
LIN {X 0,Y 524.534,Z 757.407,A -85,B 0,C 180,E1 -4646.59,E2 -4646.59} C_VEL
LIN {X 0,Y 524.913,Z 745.206,A -85,B 0,C 180,E1 -4647.367,E2 -4647.367} C_VEL
LIN {X 0,Y 525.165,Z 732.703,A -85,B 0,C 180,E1 -4647.976,E2 -4647.976} C_VEL
LIN {X 0,Y 525.325,Z 720.267,A -85,B 0,C 180,E1 -4648.41,E2 -4648.41} C_VEL
LIN {X 0,Y 525.525,Z 707.837,A -85,B 0,C 180,E1 -4648.691,E2 -4648.691} C_VEL
LIN {X 0,Y 525.943,Z 614.284,A -85,B 0,C 180,E1 -4649.983,E2 -4649.983} C_VEL
LIN {X 0,Y 524.158,Z 604.294,A -85,B 0,C 180,E1 -4650.175,E2 -4650.175} C_VEL
LIN {X 0,Y 524.486,Z 589.136,A -85,B 0,C 180,E1 -4653.328,E2 -4653.328} C_VEL
LIN {X 0,Y 523.993,Z 585.218,A -85,B 0,C 180,E1 -4654.201,E2 -4654.201} C_VEL
LIN {X 0,Y 523.906,Z 585.224,A -85,B 0,C 180,E1 -4657.107,E2 -4657.107} C_VEL
LIN {X 0,Y 523.968,Z 585.214,A -85,B 0,C 180,E1 -4659.866,E2 -4659.866} C_VEL
LIN {X 0,Y 523.96,Z 585.22,A -85,B 0,C 180,E1 -4662.837,E2 -4662.837} C_VEL
LIN {X 0,Y 523.965,Z 585.215,A -85,B 0,C 180,E1 -4665.236,E2 -4665.236} C_VEL
LIN {X 0,Y 524.001,Z 585.213,A -85,B 0,C 180,E1 -4668.394,E2 -4668.394} C_VEL
LIN {X 0,Y 524,Z 585.21,A -85,B 0,C 180,E1 -4671.516,E2 -4671.516} C_VEL
LIN {X 0,Y 524.094,Z 585.204,A -85,B 0,C 180,E1 -4674.614,E2 -4674.614} C_VEL
LIN {X 0,Y 524.103,Z 585.196,A -85,B 0,C 180,E1 -4677.695,E2 -4677.695} C_VEL
LIN {X 0,Y 524.116,Z 585.202,A -85,B 0,C 180,E1 -4680.769,E2 -4680.769} C_VEL
LIN {X 0,Y 524.069,Z 585.205,A -85,B 0,C 180,E1 -4683.075,E2 -4683.075} C_VEL
LIN {X 0,Y 524.043,Z 585.203,A -85,B 0,C 180,E1 -4686.159,E2 -4686.159} C_VEL
LIN {X 0,Y 523.997,Z 585.213,A -85,B 0,C 180,E1 -4689.262,E2 -4689.262} C_VEL
LIN {X 0,Y 524.015,Z 585.207,A -85,B 0,C 180,E1 -4691.752,E2 -4691.752} C_VEL
LIN {X 0,Y 523.983,Z 585.219,A -85,B 0,C 180,E1 -4695.053,E2 -4695.053} C_VEL
LIN {X 0,Y 523.956,Z 585.214,A -85,B 0,C 180,E1 -4697.97,E2 -4697.97} C_VEL
LIN {X 0,Y 523.964,Z 585.213,A -85,B 0,C 180,E1 -4700.411,E2 -4700.411} C_VEL
LIN {X 0,Y 523.909,Z 585.224,A -85,B 0,C 180,E1 -4702.894,E2 -4702.894} C_VEL
LIN {X 0,Y 523.947,Z 585.219,A -85,B 0,C 180,E1 -4705.419,E2 -4705.419} C_VEL
LIN {X 0,Y 523.964,Z 585.212,A -85,B 0,C 180,E1 -4708,E2 -4708} C_VEL
LIN {X 0,Y 523.946,Z 585.217,A -85,B 0,C 180,E1 -4710.857,E2 -4710.857} C_VEL
LIN {X 0,Y 523.957,Z 585.216,A -85,B 0,C 180,E1 -4713.736,E2 -4713.736} C_VEL
LIN {X 0,Y 523.917,Z 585.218,A -85,B 0,C 180,E1 -4716.405,E2 -4716.405} C_VEL
LIN {X 0,Y 523.922,Z 585.222,A -85,B 0,C 180,E1 -4719.085,E2 -4719.085} C_VEL
LIN {X 0,Y 523.953,Z 585.215,A -85,B 0,C 180,E1 -4722.119,E2 -4722.119} C_VEL
LIN {X 0,Y 523.952,Z 585.222,A -85,B 0,C 180,E1 -4725.31,E2 -4725.31} C_VEL
LIN {X 0,Y 523.969,Z 585.213,A -85,B 0,C 180,E1 -4728.689,E2 -4728.689} C_VEL
LIN {X 0,Y 523.923,Z 585.221,A -85,B 0,C 180,E1 -4731.08,E2 -4731.08} C_VEL
LIN {X 0,Y 523.929,Z 585.224,A -85,B 0,C 180,E1 -4733.829,E2 -4733.829} C_VEL
LIN {X 0,Y 523.942,Z 585.218,A -85,B 0,C 180,E1 -4736.637,E2 -4736.637} C_VEL
LIN {X 0,Y 523.955,Z 585.219,A -85,B 0,C 180,E1 -4739.357,E2 -4739.357} C_VEL
LIN {X 0,Y 523.977,Z 585.216,A -85,B 0,C 180,E1 -4742.282,E2 -4742.282} C_VEL
LIN {X 0,Y 524.034,Z 585.305,A -85,B 0,C 180,E1 -4744.878,E2 -4744.878} C_VEL
LIN {X 0,Y 525.624,Z 594.334,A -85,B 0,C 180,E1 -4746.352,E2 -4746.352} C_VEL
LIN {X 0,Y 525.28,Z 610.648,A -85,B 0,C 180,E1 -4748.824,E2 -4748.824} C_VEL
LIN {X 0,Y 524.838,Z 629.914,A -85,B 0,C 180,E1 -4751.699,E2 -4751.699} C_VEL
LIN {X 0,Y 524.387,Z 651.243,A -85,B 0,C 180,E1 -4754.846,E2 -4754.846} C_VEL
LIN {X 0,Y 525.956,Z 661.608,A -85,B 0,C 180,E1 -4755.034,E2 -4755.034} C_VEL
LIN {X 0,Y 525.535,Z 759.717,A -85,B 0,C 180,E1 -4756.392,E2 -4756.392} C_VEL
LIN {X 0,Y 525.301,Z 773.058,A -85,B 0,C 180,E1 -4756.731,E2 -4756.731} C_VEL
LIN {X 0,Y 525.072,Z 786.405,A -85,B 0,C 180,E1 -4757.241,E2 -4757.241} C_VEL
LIN {X 0,Y 524.814,Z 798.749,A -85,B 0,C 180,E1 -4757.895,E2 -4757.895} C_VEL
LIN {X 0,Y 524.505,Z 810.487,A -85,B 0,C 180,E1 -4758.699,E2 -4758.699} C_VEL
LIN {X 0,Y 524.234,Z 820.648,A -85,B 0,C 180,E1 -4759.573,E2 -4759.573} C_VEL
LIN {X 0,Y 523.975,Z 829.787,A -85,B 0,C 180,E1 -4760.543,E2 -4760.543} C_VEL
LIN {X 0,Y 523.759,Z 838.689,A -85,B 0,C 180,E1 -4761.707,E2 -4761.707} C_VEL
LIN {X 0,Y 523.584,Z 845.849,A -85,B 0,C 180,E1 -4762.868,E2 -4762.868} C_VEL
LIN {X 0,Y 523.544,Z 852.367,A -85,B 0,C 180,E1 -4764.222,E2 -4764.222} C_VEL
LIN {X 0,Y 523.361,Z 856.677,A -85,B 0,C 180,E1 -4765.379,E2 -4765.379} C_VEL
LIN {X 0,Y 523.444,Z 858.958,A -85,B 0,C 180,E1 -4766.151,E2 -4766.151} C_VEL
LIN {X 0,Y 523.368,Z 860.807,A -85,B 0,C 180,E1 -4766.921,E2 -4766.921} C_VEL
LIN {X 0,Y 523.334,Z 862.193,A -85,B 0,C 180,E1 -4767.691,E2 -4767.691} C_VEL
LIN {X 0,Y 523.25,Z 863.786,A -85,B 0,C 180,E1 -4769.23,E2 -4769.23} C_VEL
LIN {X 0,Y 523.246,Z 864,A -85,B 0,C 180,E1 -4770,E2 -4770} C_VEL
LIN {X 0,Y 523.274,Z 863.184,A -85,B 0,C 180,E1 -4771.539,E2 -4771.539} C_VEL
LIN {X 0,Y 523.334,Z 862.196,A -85,B 0,C 180,E1 -4772.309,E2 -4772.309} C_VEL
LIN {X 0,Y 523.368,Z 860.81,A -85,B 0,C 180,E1 -4773.079,E2 -4773.079} C_VEL
LIN {X 0,Y 523.442,Z 857.895,A -85,B 0,C 180,E1 -4774.235,E2 -4774.235} C_VEL
LIN {X 0,Y 523.464,Z 853.948,A -85,B 0,C 180,E1 -4775.393,E2 -4775.393} C_VEL
LIN {X 0,Y 523.523,Z 848.729,A -85,B 0,C 180,E1 -4776.58,E2 -4776.58} C_VEL
LIN {X 0,Y 523.665,Z 842.467,A -85,B 0,C 180,E1 -4777.713,E2 -4777.713} C_VEL
LIN {X 0,Y 523.857,Z 834.479,A -85,B 0,C 180,E1 -4778.875,E2 -4778.875} C_VEL
LIN {X 0,Y 524.107,Z 826.335,A -85,B 0,C 180,E1 -4779.844,E2 -4779.844} C_VEL
LIN {X 0,Y 524.366,Z 816.399,A -85,B 0,C 180,E1 -4780.815,E2 -4780.815} C_VEL
LIN {X 0,Y 524.663,Z 805.187,A -85,B 0,C 180,E1 -4781.688,E2 -4781.688} C_VEL
LIN {X 0,Y 524.921,Z 794.136,A -85,B 0,C 180,E1 -4782.369,E2 -4782.369} C_VEL
LIN {X 0,Y 525.191,Z 781.877,A -85,B 0,C 180,E1 -4782.952,E2 -4782.952} C_VEL
LIN {X 0,Y 525.386,Z 769.01,A -85,B 0,C 180,E1 -4783.39,E2 -4783.39} C_VEL
LIN {X 0,Y 525.567,Z 755.363,A -85,B 0,C 180,E1 -4783.681,E2 -4783.681} C_VEL
LIN {X 0,Y 525.88,Z 660.781,A -85,B 0,C 180,E1 -4784.98,E2 -4784.98} C_VEL
LIN {X 0,Y 524.371,Z 651.181,A -85,B 0,C 180,E1 -4785.174,E2 -4785.174} C_VEL
LIN {X 0,Y 524.866,Z 630.056,A -85,B 0,C 180,E1 -4788.3,E2 -4788.3} C_VEL
LIN {X 0,Y 525.375,Z 608.163,A -85,B 0,C 180,E1 -4791.584,E2 -4791.584} C_VEL
LIN {X 0,Y 525.681,Z 594.614,A -85,B 0,C 180,E1 -4793.645,E2 -4793.645} C_VEL
LIN {X 0,Y 524,Z 585.214,A -85,B 0,C 180,E1 -4795.203,E2 -4795.203} C_VEL
LIN {X 0,Y 523.97,Z 585.219,A -85,B 0,C 180,E1 -4797.998,E2 -4797.998} C_VEL
LIN {X 0,Y 523.944,Z 585.219,A -85,B 0,C 180,E1 -4800.854,E2 -4800.854} C_VEL
LIN {X 0,Y 523.961,Z 585.213,A -85,B 0,C 180,E1 -4803.734,E2 -4803.734} C_VEL
LIN {X 0,Y 523.924,Z 585.225,A -85,B 0,C 180,E1 -4806.404,E2 -4806.404} C_VEL
LIN {X 0,Y 523.929,Z 585.218,A -85,B 0,C 180,E1 -4809.083,E2 -4809.083} C_VEL
LIN {X 0,Y 523.969,Z 585.212,A -85,B 0,C 180,E1 -4811.311,E2 -4811.311} C_VEL
LIN {X 0,Y 523.952,Z 585.222,A -85,B 0,C 180,E1 -4814.69,E2 -4814.69} C_VEL
LIN {X 0,Y 523.953,Z 585.214,A -85,B 0,C 180,E1 -4817.881,E2 -4817.881} C_VEL
LIN {X 0,Y 523.919,Z 585.225,A -85,B 0,C 180,E1 -4820.915,E2 -4820.915} C_VEL
LIN {X 0,Y 523.922,Z 585.217,A -85,B 0,C 180,E1 -4823.827,E2 -4823.827} C_VEL
LIN {X 0,Y 523.937,Z 585.221,A -85,B 0,C 180,E1 -4826.635,E2 -4826.635} C_VEL
LIN {X 0,Y 523.957,Z 585.216,A -85,B 0,C 180,E1 -4829.355,E2 -4829.355} C_VEL
LIN {X 0,Y 523.973,Z 585.212,A -85,B 0,C 180,E1 -4832.28,E2 -4832.28} C_VEL
LIN {X 0,Y 523.947,Z 585.217,A -85,B 0,C 180,E1 -4834.581,E2 -4834.581} C_VEL
LIN {X 0,Y 523.909,Z 585.228,A -85,B 0,C 180,E1 -4837.106,E2 -4837.106} C_VEL
LIN {X 0,Y 523.97,Z 585.212,A -85,B 0,C 180,E1 -4839.865,E2 -4839.865} C_VEL
LIN {X 0,Y 523.962,Z 585.217,A -85,B 0,C 180,E1 -4842.837,E2 -4842.837} C_VEL
LIN {X 0,Y 523.967,Z 585.221,A -85,B 0,C 180,E1 -4845.235,E2 -4845.235} C_VEL
